            if (move_thread_flag_427 > 1):
              join move_thread_han_427
              $ 428 "Until (distance)"
              break
            end
            sync()
          end
          $ 429 "MoveJ"
          $ 430 "internos" "breakAfter"
          movej(internos, a=0.6981317007977318, v=0.5235987755982988)
          $ 431 "Wait: 0.3"
          sleep(0.3)
          $ 432 "Set CO[1]=Apagar"
          set_configurable_digital_out(1, False)
          $ 433 "Wait: 0.3"
          sleep(0.3)
          $ 434 "If barrenoActual≟13"
          if (barrenoActual == 13):
            $ 435 "Direction: Base Z+"
            global move_thread_flag_435=0
            thread move_thread_435():
              enter_critical
              move_thread_flag_435 = 1
              local towardsPos=calculate_point_to_move_towards(p[0.0,0.0,0.0,0.0,0.0,0.0], [0.0,0.0,1.0], 0.03)
              movel(towardsPos, a=1.2, v=0.25)
              move_thread_flag_435 = 2
              exit_critical
            end
            move_thread_flag_435 = 0
            move_thread_han_435 = run move_thread_435()
            while (True):
              sleep(1.0E-10)
              if (move_thread_flag_435 > 1):
                join move_thread_han_435
                $ 436 "Until (distance)"
                break
              end
              sync()
            end
            $ 437 "MoveJ"
            $ 438 "Zona_der1" "breakAfter"
            movej(get_inverse_kin(Zona_der1_p, qnear=Zona_der1_q), a=1.3962634015954636, v=1.0471975511965976)
            $ 439 "Posicion_Cero" "breakAfter"
            movej(get_inverse_kin(Posicion_Cero_p, qnear=Posicion_Cero_q), a=1.3962634015954636, v=1.0471975511965976)
            $ 440 "Call Quitar_Broca_Chida"
            Quitar_Broca_Chida()
            $ 441 "Call Poner_Broca"
            Poner_Broca()
            $ 442 "MoveJ"
            $ 443 "Posicion_Cero" "breakAfter"
            movej(get_inverse_kin(Posicion_Cero_p, qnear=Posicion_Cero_q), a=1.3962634015954636, v=1.0471975511965976)
            $ 444 "Zona_der1" "breakAfter"
            movej(get_inverse_kin(Zona_der1_p, qnear=Zona_der1_q), a=1.3962634015954636, v=1.0471975511965976)
          else:
            $ 445 "ElseIf barrenoActual≟27"
            if (barrenoActual == 27):
              $ 446 "Direction: Base Z+"
              global move_thread_flag_446=0
              thread move_thread_446():
                enter_critical
                move_thread_flag_446 = 1
                local towardsPos=calculate_point_to_move_towards(p[0.0,0.0,0.0,0.0,0.0,0.0], [0.0,0.0,1.0], 0.03)
                movel(towardsPos, a=1.2, v=0.25)
                move_thread_flag_446 = 2
                exit_critical
              end
              move_thread_flag_446 = 0
              move_thread_han_446 = run move_thread_446()
              while (True):
                sleep(1.0E-10)
                if (move_thread_flag_446 > 1):
                  join move_thread_han_446
                  $ 447 "Until (distance)"
                  break
                end
                sync()
              end
              $ 448 "MoveJ"
              $ 449 "Zona_der1" "breakAfter"
              movej(get_inverse_kin(Zona_der1_p, qnear=Zona_der1_q), a=1.3962634015954636, v=1.0471975511965976)
              $ 450 "Posicion_Cero" "breakAfter"
              movej(get_inverse_kin(Posicion_Cero_p, qnear=Posicion_Cero_q), a=1.3962634015954636, v=1.0471975511965976)
              $ 451 "Call Quitar_Broca_Chida"
              Quitar_Broca_Chida()
              $ 452 "Set carrusel_home=Encender"
              modbus_set_output_signal("carrusel_home", True)
              $ 453 "Wait: 1.0"
              sleep(1.0)
              $ 454 "Set carrusel_home=Apagar"
              modbus_set_output_signal("carrusel_home", False)
              $ 455 "Set mensaje_mw10=70"
              modbus_set_output_register("mensaje_mw10", 70)
              $ 456 "Wait Continuar_M30=HI"
              while (modbus_get_signal_status("Continuar_M30") == False):
                sync()
              end
              $ 457 "Wait: 1.0"
              sleep(1.0)
              $ 458 "Set mensaje_mw10=120"
              modbus_set_output_register("mensaje_mw10", 120)
              $ 459 "Wait Continuar_M30=HI"
              while (modbus_get_signal_status("Continuar_M30") == False):
                sync()
              end
              $ 460 "Wait: 1.0"
              sleep(1.0)
              $ 461 "Set carrusel_home=Encender"
              modbus_set_output_signal("carrusel_home", True)
              $ 462 "Wait: 1.0"
              sleep(1.0)
              $ 463 "Set carrusel_home=Apagar"
              modbus_set_output_signal("carrusel_home", False)
              $ 464 "Set mensaje_mw10=75"
              modbus_set_output_register("mensaje_mw10", 75)
              $ 465 "Wait Continuar_M30=HI"
              while (modbus_get_signal_status("Continuar_M30") == False):
                sync()
              end
              $ 466 "Wait: 1.0"
              sleep(1.0)
              $ 467 "Call Poner_Broca"
              Poner_Broca()
              $ 468 "broca≔1935"
              global broca=1935
              $ 469 "MoveJ"
              $ 470 "Posicion_Cero" "breakAfter"
              movej(get_inverse_kin(Posicion_Cero_p, qnear=Posicion_Cero_q), a=1.3962634015954636, v=1.0471975511965976)
              $ 471 "Zona_der1" "breakAfter"
              movej(get_inverse_kin(Zona_der1_p, qnear=Zona_der1_q), a=1.3962634015954636, v=1.0471975511965976)
              $ 472 "Set mensaje_mw10=80"
              modbus_set_output_register("mensaje_mw10", 80)
              $ 473 "Wait Continuar_M30=HI"
              while (modbus_get_signal_status("Continuar_M30") == False):
                sync()
              end
              $ 474 "Wait: 1.0"
              sleep(1.0)
              $ 475 "Set mensaje_mw10=150"
              modbus_set_output_register("mensaje_mw10", 150)
              $ 476 "Wait Continuar_M30=HI"
              while (modbus_get_signal_status("Continuar_M30") == False):
                sync()
              end
              $ 477 "Wait: 1.0"
              sleep(1.0)
            end
          end
          $ 478 "barrenoActual≔barrenoActual+1"
          global barrenoActual=barrenoActual+1
        end
        $ 479 "Linea 1 a 1935"
        $ 480 "broca≔1935"
        global broca=1935
        $ 481 "Buje_inicial"
        $ 482 "Buje_Inicial≔L1B2"
        global Buje_Inicial=L1B2
        $ 483 "Buje_final"
        $ 484 "Buje_Final≔L1B1"
        global Buje_Final=L1B1
        $ 485 "barrenosTotales≔27"
        global barrenosTotales=27
        $ 486 "barrenoActual≔1"
        global barrenoActual=1
        $ 487 "Loop barrenoActual≤barrenosTotales"
        while (barrenoActual <= barrenosTotales):
          $ 488 "MoveL"
          $ 489 "bajada_broca≔p[0,0,0.009,0,0,0]"
          global bajada_broca=p[0,0,0.009,0,0,0]
          $ 490 "internos≔interpolate_pose(Buje_Inicial, Buje_Final, ((barrenoActual)-1)/((barrenosTotales)-1))"
          global internos= interpolate_pose (Buje_Inicial, Buje_Final, ((barrenoActual)-1)/((barrenosTotales)-1))
          $ 491 "Alturas"
          $ 492 "If barrenoActual≟1 or barrenoActual≟3 or barrenoActual≟5 or barrenoActual≟7 or barrenoActual≟9 or barrenoActual≟11 or barrenoActual≟13 or barrenoActual≟15 or barrenoActual≟17 or barrenoActual≟19 or barrenoActual≟21 or barrenoActual≟23 or barrenoActual≟25 or barrenoActual≟27"
          if (barrenoActual == 1  or  barrenoActual == 3  or  barrenoActual == 5  or  barrenoActual == 7  or  barrenoActual == 9  or  barrenoActual == 11  or  barrenoActual == 13  or  barrenoActual == 15  or  barrenoActual == 17  or  barrenoActual == 19  or  barrenoActual == 21  or  barrenoActual == 23  or  barrenoActual == 25  or  barrenoActual == 27):
            $ 493 "Set mensaje_mw10=200"
            modbus_set_output_register("mensaje_mw10", 200)
            $ 494 "Wait Continuar_M30=HI"
            while (modbus_get_signal_status("Continuar_M30") == False):
              sync()
            end
            $ 495 "Wait: 1.0"
            sleep(1.0)
            $ 496 "Set mensaje_mw10=150"
            modbus_set_output_register("mensaje_mw10", 150)
            $ 497 "Wait: 1.0"
            sleep(1.0)
          end
          $ 498 "MoveJ"
          $ 499 "internos" "breakAfter"
          movej(internos, a=0.6981317007977318, v=0.5235987755982988)
          $ 500 "Wait: 2.0"
          sleep(2.0)
          $ 501 "If P1h[2]<P2h[2]"
          if (P1h[2]<P2h[2]):
            $ 502 "acomodo≔(altura/(barrenosTotales-1))*(barrenoActual-1)"
            global acomodo=(altura/(barrenosTotales-1))*(barrenoActual-1)
            $ 503 "tcp≔get_actual_tcp_pose()"
            global tcp= get_actual_tcp_pose ()
            $ 504 "offset_altura≔p[tcp[0],tcp[1],((alta-0.0095)-(acomodo/1000)),tcp[3],tcp[4],tcp[5]]"
            global offset_altura=p[tcp[0],tcp[1],((alta-0.0095)-(acomodo/1000)),tcp[3],tcp[4],tcp[5]]
            $ 505 "MoveL"
            $ 506 "offset_altura" "breakAfter"
            movel(offset_altura, a=0.04, v=0.03)
          else:
            $ 507 "Else" "noBreak"
            $ 508 "acomodo≔(altura/(barrenosTotales-1))*(26-(barrenoActual-1))"
            global acomodo=(altura/(barrenosTotales-1))*(26-(barrenoActual-1))
            $ 509 "tcp≔get_actual_tcp_pose()"
            global tcp= get_actual_tcp_pose ()
            $ 510 "offset_altura≔p[tcp[0],tcp[1],((alta-0.0095)-(acomodo/1000)),tcp[3],tcp[4],tcp[5]]"
            global offset_altura=p[tcp[0],tcp[1],((alta-0.0095)-(acomodo/1000)),tcp[3],tcp[4],tcp[5]]
            $ 511 "MoveL"
            $ 512 "offset_altura" "breakAfter"
            movel(offset_altura, a=0.04, v=0.03)
          end
          $ 513 "Freemove"
          $ 514 "Wait: 2.0"
          sleep(2.0)
          $ 515 "freedrive_mode()"
          freedrive_mode()
          $ 516 "Wait: 2.5"
          sleep(2.5)
          $ 517 "end_freedrive_mode()"
          end_freedrive_mode()
          $ 518 "Wait: 0.3"
          sleep(0.3)
          $ 519 "Set CO[1]=Encender"
          set_configurable_digital_out(1, True)
          $ 520 "Wait: 1.0"
          sleep(1.0)
          $ 521 "Wait: 0.3"
          sleep(0.3)
          $ 522 "Wait: 0.3"
          sleep(0.3)
          $ 523 "Wait: 0.3"
          sleep(0.3)
          $ 524 "Loop 2 times"
          Loop_63 = 0
          while (Loop_63 < 2):
            $ 525 "Poses_taladrado≔pose_sub(get_actual_tcp_pose(), bajada_broca)"
            global Poses_taladrado= pose_sub ( get_actual_tcp_pose (), bajada_broca)
            $ 526 "Poses_taladrado" "breakAfter"
            movel(Poses_taladrado, a=0.005, v=0.001)
            $ 527 "If bajada_broca≟p[0,0,0.018,0,0,0]"
            if (bajada_broca == p[0,0,0.018,0,0,0]):
              $ 528 "num_barreno≔str_cat('Barreno: ',barrenoActual)"
              global num_barreno=str_cat("Barreno: ",barrenoActual)
              $ 529 "tcp_actual≔get_actual_tcp_pose()"
              global tcp_actual= get_actual_tcp_pose ()
              $ 530 "X_actual≔str_cat('     X: ',tcp_actual[0])"
              global X_actual=str_cat("     X: ",tcp_actual[0])
              $ 531 "Y_actual≔str_cat('     Y: ',tcp_actual[1])"
              global Y_actual=str_cat("     Y: ",tcp_actual[1])
              $ 532 "pos_barreno≔str_cat(X_actual,Y_actual)"
              global pos_barreno=str_cat(X_actual,Y_actual)
              $ 533 "textmsg(num_barreno,pos_barreno)"
              textmsg(num_barreno,pos_barreno)
            end
            $ 534 "Poses_taladrado≔pose_add(get_actual_tcp_pose(), bajada_broca)"
            global Poses_taladrado= pose_add ( get_actual_tcp_pose (), bajada_broca)
            $ 535 "Poses_taladrado" "breakAfter"
            movel(Poses_taladrado, a=0.01, v=0.01)
            $ 536 "bajada_broca≔pose_add(bajada_broca, p[0,0,0.009,0,0,0])"
            global bajada_broca= pose_add (bajada_broca, p[0,0,0.009,0,0,0])
            Loop_63 = Loop_63 + 1
          end
          $ 537 "Direction: Base Z+"
          global move_thread_flag_537=0
          thread move_thread_537():
            enter_critical
            move_thread_flag_537 = 1
            local towardsPos=calculate_point_to_move_towards(p[0.0,0.0,0.0,0.0,0.0,0.0], [0.0,0.0,1.0], 0.05)
            movel(towardsPos, a=0.01, v=0.01)
            move_thread_flag_537 = 2
            exit_critical
          end
          move_thread_flag_537 = 0
          move_thread_han_537 = run move_thread_537()
          while (True):
            sleep(1.0E-10)
            if (move_thread_flag_537 > 1):
              join move_thread_han_537
              $ 538 "Until (distance)"
              break
            end
            sync()
          end
          $ 539 "MoveJ"
          $ 540 "internos" "breakAfter"
          movej(internos, a=0.6981317007977318, v=0.5235987755982988)
          $ 541 "Wait: 0.3"
          sleep(0.3)
          $ 542 "Set CO[1]=Apagar"
          set_configurable_digital_out(1, False)
          $ 543 "Wait: 0.3"
          sleep(0.3)
          $ 544 "If barrenoActual≟13 or barrenoActual≟27"
          if (barrenoActual == 13  or  barrenoActual == 27):
            $ 545 "Direction: Base Z+"
            global move_thread_flag_545=0
            thread move_thread_545():
              enter_critical
              move_thread_flag_545 = 1
              local towardsPos=calculate_point_to_move_towards(p[0.0,0.0,0.0,0.0,0.0,0.0], [0.0,0.0,1.0], 0.03)
              movel(towardsPos, a=0.04, v=0.03)
              move_thread_flag_545 = 2
              exit_critical
            end
            move_thread_flag_545 = 0
            move_thread_han_545 = run move_thread_545()
            while (True):
              sleep(1.0E-10)
              if (move_thread_flag_545 > 1):
                join move_thread_han_545
                $ 546 "Until (distance)"
                break
              end
              sync()
            end
            $ 547 "MoveJ"
            $ 548 "Zona_der1" "breakAfter"
            movej(get_inverse_kin(Zona_der1_p, qnear=Zona_der1_q), a=0.6981317007977318, v=0.5235987755982988)
            $ 549 "Posicion_Cero" "breakAfter"
            movej(get_inverse_kin(Posicion_Cero_p, qnear=Posicion_Cero_q), a=0.6981317007977318, v=0.5235987755982988)
            $ 550 "Call Quitar_Broca_Chida"
            Quitar_Broca_Chida()
            $ 551 "If barrenoActual≟13"
            if (barrenoActual == 13):
              $ 552 "Call Poner_Broca"
              Poner_Broca()
            else:
              $ 553 "ElseIf barrenoActual≟27"
              if (barrenoActual == 27):
                $ 554 "Call Poner_Broca"
                Poner_Broca()
              end
            end
            $ 555 "MoveJ"
            $ 556 "Posicion_Cero" "breakAfter"
            movej(get_inverse_kin(Posicion_Cero_p, qnear=Posicion_Cero_q), a=0.6981317007977318, v=0.5235987755982988)
            $ 557 "Zona_der1" "breakAfter"
            movej(get_inverse_kin(Zona_der1_p, qnear=Zona_der1_q), a=0.6981317007977318, v=0.5235987755982988)
          end
          $ 558 "barrenoActual≔barrenoActual+1"
          global barrenoActual=barrenoActual+1
        end
        $ 559 "Linea 2 a 1935"
        $ 560 "broca≔1935"
        global broca=1935
        $ 561 "Buje_inicial"
        $ 562 "Buje_Inicial≔L2B2"
        global Buje_Inicial=L2B2
        $ 563 "Buje_final"
        $ 564 "Buje_Final≔L2B1"
        global Buje_Final=L2B1
        $ 565 "barrenosTotales≔27"
        global barrenosTotales=27
        $ 566 "barrenoActual≔1"
        global barrenoActual=1
        $ 567 "Loop barrenoActual≤barrenosTotales"
        while (barrenoActual <= barrenosTotales):
          $ 568 "MoveL"
          $ 569 "bajada_broca≔p[0,0,0.009,0,0,0]"
          global bajada_broca=p[0,0,0.009,0,0,0]
          $ 570 "internos≔interpolate_pose(Buje_Inicial, Buje_Final, ((barrenoActual)-1)/((barrenosTotales)-1))"
          global internos= interpolate_pose (Buje_Inicial, Buje_Final, ((barrenoActual)-1)/((barrenosTotales)-1))
          $ 571 "Alturas"
          $ 572 "If barrenoActual≟1 or barrenoActual≟3 or barrenoActual≟5 or barrenoActual≟7 or barrenoActual≟9 or barrenoActual≟11 or barrenoActual≟13 or barrenoActual≟15 or barrenoActual≟17 or barrenoActual≟19 or barrenoActual≟21 or barrenoActual≟23 or barrenoActual≟25 or barrenoActual≟27"
          if (barrenoActual == 1  or  barrenoActual == 3  or  barrenoActual == 5  or  barrenoActual == 7  or  barrenoActual == 9  or  barrenoActual == 11  or  barrenoActual == 13  or  barrenoActual == 15  or  barrenoActual == 17  or  barrenoActual == 19  or  barrenoActual == 21  or  barrenoActual == 23  or  barrenoActual == 25  or  barrenoActual == 27):
            $ 573 "Set mensaje_mw10=200"
            modbus_set_output_register("mensaje_mw10", 200)
            $ 574 "Wait Continuar_M30=HI"
            while (modbus_get_signal_status("Continuar_M30") == False):
              sync()
            end
            $ 575 "Wait: 1.0"
            sleep(1.0)
            $ 576 "Set mensaje_mw10=150"
            modbus_set_output_register("mensaje_mw10", 150)
            $ 577 "Wait: 1.0"
            sleep(1.0)
          end
          $ 578 "MoveJ"
          $ 579 "internos" "breakAfter"
          movej(internos, a=0.6981317007977318, v=0.5235987755982988)
          $ 580 "Wait: 2.0"
          sleep(2.0)
          $ 581 "If P1h[2]<P2h[2]"
          if (P1h[2]<P2h[2]):
            $ 582 "acomodo≔(altura/(barrenosTotales-1))*(barrenoActual-1)"
            global acomodo=(altura/(barrenosTotales-1))*(barrenoActual-1)
            $ 583 "tcp≔get_actual_tcp_pose()"
            global tcp= get_actual_tcp_pose ()
            $ 584 "offset_altura≔p[tcp[0],tcp[1],((alta-0.0095)-(acomodo/1000)),tcp[3],tcp[4],tcp[5]]"
            global offset_altura=p[tcp[0],tcp[1],((alta-0.0095)-(acomodo/1000)),tcp[3],tcp[4],tcp[5]]
            $ 585 "MoveL"
            $ 586 "offset_altura" "breakAfter"
            movel(offset_altura, a=0.04, v=0.03)
          else:
            $ 587 "Else" "noBreak"
            $ 588 "acomodo≔(altura/(barrenosTotales-1))*(26-(barrenoActual-1))"
            global acomodo=(altura/(barrenosTotales-1))*(26-(barrenoActual-1))
            $ 589 "tcp≔get_actual_tcp_pose()"
            global tcp= get_actual_tcp_pose ()
            $ 590 "offset_altura≔p[tcp[0],tcp[1],((alta-0.0095)-(acomodo/1000)),tcp[3],tcp[4],tcp[5]]"
            global offset_altura=p[tcp[0],tcp[1],((alta-0.0095)-(acomodo/1000)),tcp[3],tcp[4],tcp[5]]
            $ 591 "MoveL"
            $ 592 "offset_altura" "breakAfter"
            movel(offset_altura, a=0.04, v=0.03)
          end
          $ 593 "Freemove"
          $ 594 "Wait: 2.0"
          sleep(2.0)
          $ 595 "freedrive_mode()"
          freedrive_mode()
          $ 596 "Wait: 2.5"
          sleep(2.5)
          $ 597 "end_freedrive_mode()"
          end_freedrive_mode()
          $ 598 "Wait: 0.3"
          sleep(0.3)
          $ 599 "Set CO[1]=Encender"
          set_configurable_digital_out(1, True)
          $ 600 "Wait: 1.0"
          sleep(1.0)
          $ 601 "Wait: 0.3"
          sleep(0.3)
          $ 602 "Wait: 0.3"
          sleep(0.3)
          $ 603 "Wait: 0.3"
          sleep(0.3)
          $ 604 "Loop 2 times"
          Loop_65 = 0
          while (Loop_65 < 2):
            $ 605 "Poses_taladrado≔pose_sub(get_actual_tcp_pose(), bajada_broca)"
            global Poses_taladrado= pose_sub ( get_actual_tcp_pose (), bajada_broca)
            $ 606 "Poses_taladrado" "breakAfter"
            movel(Poses_taladrado, a=0.005, v=0.001)
            $ 607 "If bajada_broca≟p[0,0,0.018,0,0,0]"
            if (bajada_broca == p[0,0,0.018,0,0,0]):
              $ 608 "num_barreno≔str_cat('Barreno: ',barrenoActual)"
              global num_barreno=str_cat("Barreno: ",barrenoActual)
              $ 609 "tcp_actual≔get_actual_tcp_pose()"
              global tcp_actual= get_actual_tcp_pose ()
              $ 610 "X_actual≔str_cat('     X: ',tcp_actual[0])"
              global X_actual=str_cat("     X: ",tcp_actual[0])
              $ 611 "Y_actual≔str_cat('     Y: ',tcp_actual[1])"
              global Y_actual=str_cat("     Y: ",tcp_actual[1])
              $ 612 "pos_barreno≔str_cat(X_actual,Y_actual)"
              global pos_barreno=str_cat(X_actual,Y_actual)
              $ 613 "textmsg(num_barreno,pos_barreno)"
              textmsg(num_barreno,pos_barreno)
            end
            $ 614 "Poses_taladrado≔pose_add(get_actual_tcp_pose(), bajada_broca)"
            global Poses_taladrado= pose_add ( get_actual_tcp_pose (), bajada_broca)
            $ 615 "Poses_taladrado" "breakAfter"
            movel(Poses_taladrado, a=0.01, v=0.01)
            $ 616 "bajada_broca≔pose_add(bajada_broca, p[0,0,0.009,0,0,0])"
            global bajada_broca= pose_add (bajada_broca, p[0,0,0.009,0,0,0])
            Loop_65 = Loop_65 + 1
          end
          $ 617 "Direction: Base Z+"
          global move_thread_flag_617=0
          thread move_thread_617():
            enter_critical
            move_thread_flag_617 = 1
            local towardsPos=calculate_point_to_move_towards(p[0.0,0.0,0.0,0.0,0.0,0.0], [0.0,0.0,1.0], 0.05)
            movel(towardsPos, a=0.01, v=0.01)
            move_thread_flag_617 = 2
            exit_critical
          end
          move_thread_flag_617 = 0
          move_thread_han_617 = run move_thread_617()
          while (True):
            sleep(1.0E-10)
            if (move_thread_flag_617 > 1):
              join move_thread_han_617
              $ 618 "Until (distance)"
              break
            end
            sync()
          end
          $ 619 "MoveJ"
          $ 620 "internos" "breakAfter"
          movej(internos, a=0.6981317007977318, v=0.5235987755982988)
          $ 621 "Wait: 0.3"
          sleep(0.3)
          $ 622 "Set CO[1]=Apagar"
          set_configurable_digital_out(1, False)
          $ 623 "Wait: 0.3"
          sleep(0.3)
          $ 624 "If barrenoActual≟13"
          if (barrenoActual == 13):
            $ 625 "Direction: Base Z+"
            global move_thread_flag_625=0
            thread move_thread_625():
              enter_critical
              move_thread_flag_625 = 1
              local towardsPos=calculate_point_to_move_towards(p[0.0,0.0,0.0,0.0,0.0,0.0], [0.0,0.0,1.0], 0.03)
              movel(towardsPos, a=0.04, v=0.03)
              move_thread_flag_625 = 2
              exit_critical
            end
            move_thread_flag_625 = 0
            move_thread_han_625 = run move_thread_625()
            while (True):
              sleep(1.0E-10)
              if (move_thread_flag_625 > 1):
                join move_thread_han_625
                $ 626 "Until (distance)"
                break
              end
              sync()
            end
            $ 627 "MoveJ"
            $ 628 "Zona_der1" "breakAfter"
            movej(get_inverse_kin(Zona_der1_p, qnear=Zona_der1_q), a=1.3962634015954636, v=1.0471975511965976)
            $ 629 "Posicion_Cero" "breakAfter"
            movej(get_inverse_kin(Posicion_Cero_p, qnear=Posicion_Cero_q), a=1.3962634015954636, v=1.0471975511965976)
            $ 630 "Call Quitar_Broca_Chida"
            Quitar_Broca_Chida()
            $ 631 "Call Poner_Broca"
            Poner_Broca()
            $ 632 "MoveJ"
            $ 633 "Posicion_Cero" "breakAfter"
            movej(get_inverse_kin(Posicion_Cero_p, qnear=Posicion_Cero_q), a=1.3962634015954636, v=1.0471975511965976)
            $ 634 "Zona_der1" "breakAfter"
            movej(get_inverse_kin(Zona_der1_p, qnear=Zona_der1_q), a=1.3962634015954636, v=1.0471975511965976)
          else:
            $ 635 "ElseIf barrenoActual≟27"
            if (barrenoActual == 27):
              $ 636 "Direction: Base Z+"
              global move_thread_flag_636=0
              thread move_thread_636():
                enter_critical
                move_thread_flag_636 = 1
                local towardsPos=calculate_point_to_move_towards(p[0.0,0.0,0.0,0.0,0.0,0.0], [0.0,0.0,1.0], 0.03)
                movel(towardsPos, a=0.04, v=0.03)
                move_thread_flag_636 = 2
                exit_critical
              end
              move_thread_flag_636 = 0
              move_thread_han_636 = run move_thread_636()
              while (True):
                sleep(1.0E-10)
                if (move_thread_flag_636 > 1):
                  join move_thread_han_636
                  $ 637 "Until (distance)"
                  break
                end
                sync()
              end
              $ 638 "MoveJ"
              $ 639 "Zona_der1" "breakAfter"
              movej(get_inverse_kin(Zona_der1_p, qnear=Zona_der1_q), a=1.3962634015954636, v=1.0471975511965976)
              $ 640 "Posicion_Cero" "breakAfter"
              movej(get_inverse_kin(Posicion_Cero_p, qnear=Posicion_Cero_q), a=1.3962634015954636, v=1.0471975511965976)
              $ 641 "Call Quitar_Broca_Chida"
              Quitar_Broca_Chida()
              $ 642 "Set carrusel_home=Encender"
              modbus_set_output_signal("carrusel_home", True)
              $ 643 "Wait: 1.0"
              sleep(1.0)
              $ 644 "Set carrusel_home=Apagar"
              modbus_set_output_signal("carrusel_home", False)
              $ 645 "Set mensaje_mw10=85"
              modbus_set_output_register("mensaje_mw10", 85)
              $ 646 "Wait Continuar_M30=HI"
              while (modbus_get_signal_status("Continuar_M30") == False):
                sync()
              end
              $ 647 "Wait: 1.0"
              sleep(1.0)
              $ 648 "Set mensaje_mw10=120"
              modbus_set_output_register("mensaje_mw10", 120)
              $ 649 "Wait Continuar_M30=HI"
              while (modbus_get_signal_status("Continuar_M30") == False):
                sync()
              end
              $ 650 "Wait: 1.0"
              sleep(1.0)
              $ 651 "Set carrusel_home=Encender"
              modbus_set_output_signal("carrusel_home", True)
              $ 652 "Wait: 1.0"
              sleep(1.0)
              $ 653 "Set carrusel_home=Apagar"
              modbus_set_output_signal("carrusel_home", False)
              $ 654 "Set mensaje_mw10=90"
              modbus_set_output_register("mensaje_mw10", 90)
              $ 655 "Wait Continuar_M30=HI"
              while (modbus_get_signal_status("Continuar_M30") == False):
                sync()
              end
              $ 656 "Wait: 1.0"
              sleep(1.0)
              $ 657 "Call Poner_Broca"
              Poner_Broca()
              $ 658 "broca≔217"
              global broca=217
              $ 659 "MoveJ"
              $ 660 "Posicion_Cero" "breakAfter"
              movej(get_inverse_kin(Posicion_Cero_p, qnear=Posicion_Cero_q), a=1.3962634015954636, v=1.0471975511965976)
              $ 661 "Zona_der1" "breakAfter"
              movej(get_inverse_kin(Zona_der1_p, qnear=Zona_der1_q), a=1.3962634015954636, v=1.0471975511965976)
              $ 662 "Set mensaje_mw10=95"
              modbus_set_output_register("mensaje_mw10", 95)
              $ 663 "Wait Continuar_M30=HI"
              while (modbus_get_signal_status("Continuar_M30") == False):
                sync()
              end
              $ 664 "Wait: 1.0"
              sleep(1.0)
              $ 665 "Set mensaje_mw10=150"
              modbus_set_output_register("mensaje_mw10", 150)
              $ 666 "Wait Continuar_M30=HI"
              while (modbus_get_signal_status("Continuar_M30") == False):
                sync()
              end
              $ 667 "Wait: 1.0"
              sleep(1.0)
            end
          end
          $ 668 "barrenoActual≔barrenoActual+1"
          global barrenoActual=barrenoActual+1
        end
        $ 669 "Linea 1 a 217"
        $ 670 "broca≔217"
        global broca=217
        $ 671 "Buje_inicial"
        $ 672 "Buje_Inicial≔L1B2"
        global Buje_Inicial=L1B2
        $ 673 "Buje_final"
        $ 674 "Buje_Final≔L1B1"
        global Buje_Final=L1B1
        $ 675 "barrenosTotales≔27"
        global barrenosTotales=27
        $ 676 "barrenoActual≔1"
        global barrenoActual=1
        $ 677 "Loop barrenoActual≤barrenosTotales"
        while (barrenoActual <= barrenosTotales):
          $ 678 "MoveL"
          $ 679 "bajada_broca≔p[0,0,0.018,0,0,0]"
          global bajada_broca=p[0,0,0.018,0,0,0]
          $ 680 "internos≔interpolate_pose(Buje_Inicial, Buje_Final, ((barrenoActual)-1)/((barrenosTotales)-1))"
          global internos= interpolate_pose (Buje_Inicial, Buje_Final, ((barrenoActual)-1)/((barrenosTotales)-1))
          $ 681 "Wait: 2.0"
          sleep(2.0)
          $ 682 "Alturas"
          $ 683 "If barrenoActual≟1 or barrenoActual≟3 or barrenoActual≟5 or barrenoActual≟7 or barrenoActual≟9 or barrenoActual≟11 or barrenoActual≟13 or barrenoActual≟15 or barrenoActual≟17 or barrenoActual≟19 or barrenoActual≟21 or barrenoActual≟23 or barrenoActual≟25 or barrenoActual≟27"
          if (barrenoActual == 1  or  barrenoActual == 3  or  barrenoActual == 5  or  barrenoActual == 7  or  barrenoActual == 9  or  barrenoActual == 11  or  barrenoActual == 13  or  barrenoActual == 15  or  barrenoActual == 17  or  barrenoActual == 19  or  barrenoActual == 21  or  barrenoActual == 23  or  barrenoActual == 25  or  barrenoActual == 27):
            $ 684 "Set mensaje_mw10=200"
            modbus_set_output_register("mensaje_mw10", 200)
            $ 685 "Wait Continuar_M30=HI"
            while (modbus_get_signal_status("Continuar_M30") == False):
              sync()
            end
            $ 686 "Wait: 1.0"
            sleep(1.0)
            $ 687 "Set mensaje_mw10=150"
            modbus_set_output_register("mensaje_mw10", 150)
            $ 688 "Wait: 1.0"
            sleep(1.0)
          end
          $ 689 "MoveJ"
          $ 690 "internos" "breakAfter"
          movej(internos, a=0.6981317007977318, v=0.5235987755982988)
          $ 691 "Wait: 2.0"
          sleep(2.0)
          $ 692 "If P1h[2]<P2h[2]"
          if (P1h[2]<P2h[2]):
            $ 693 "acomodo≔(altura/(barrenosTotales-1))*(barrenoActual-1)"
            global acomodo=(altura/(barrenosTotales-1))*(barrenoActual-1)
            $ 694 "tcp≔get_actual_tcp_pose()"
            global tcp= get_actual_tcp_pose ()
            $ 695 "offset_altura≔p[tcp[0],tcp[1],((alta-0.0095)-(acomodo/1000)),tcp[3],tcp[4],tcp[5]]"
            global offset_altura=p[tcp[0],tcp[1],((alta-0.0095)-(acomodo/1000)),tcp[3],tcp[4],tcp[5]]
            $ 696 "MoveL"
            $ 697 "offset_altura" "breakAfter"
            movel(offset_altura, a=0.04, v=0.03)
          else:
            $ 698 "Else" "noBreak"
            $ 699 "acomodo≔(altura/(barrenosTotales-1))*(26-(barrenoActual-1))"
            global acomodo=(altura/(barrenosTotales-1))*(26-(barrenoActual-1))
            $ 700 "tcp≔get_actual_tcp_pose()"
            global tcp= get_actual_tcp_pose ()
            $ 701 "offset_altura≔p[tcp[0],tcp[1],((alta-0.0095)-(acomodo/1000)),tcp[3],tcp[4],tcp[5]]"
            global offset_altura=p[tcp[0],tcp[1],((alta-0.0095)-(acomodo/1000)),tcp[3],tcp[4],tcp[5]]
            $ 702 "MoveL"
            $ 703 "offset_altura" "breakAfter"
            movel(offset_altura, a=0.04, v=0.03)
          end
          $ 704 "Freemove"
          $ 705 "Wait: 2.0"
          sleep(2.0)
          $ 706 "freedrive_mode()"
          freedrive_mode()
          $ 707 "Wait: 2.5"
          sleep(2.5)
          $ 708 "end_freedrive_mode()"
          end_freedrive_mode()
          $ 709 "Wait: 0.3"
          sleep(0.3)
          $ 710 "Set CO[1]=Encender"
          set_configurable_digital_out(1, True)
          $ 711 "Wait: 1.0"
          sleep(1.0)
          $ 712 "Wait: 0.3"
          sleep(0.3)
          $ 713 "Wait: 0.3"
          sleep(0.3)
          $ 714 "Wait: 0.3"
          sleep(0.3)
          $ 715 "Loop 1 times"
          Loop_67 = 0
          while (Loop_67 < 1):
            $ 716 "Poses_taladrado≔pose_sub(get_actual_tcp_pose(), bajada_broca)"
            global Poses_taladrado= pose_sub ( get_actual_tcp_pose (), bajada_broca)
            $ 717 "Poses_taladrado" "breakAfter"
            movel(Poses_taladrado, a=0.005, v=0.001)
            $ 718 "If bajada_broca≟p[0,0,0.018,0,0,0]"
            if (bajada_broca == p[0,0,0.018,0,0,0]):
              $ 719 "num_barreno≔str_cat('Barreno: ',barrenoActual)"
              global num_barreno=str_cat("Barreno: ",barrenoActual)
              $ 720 "tcp_actual≔get_actual_tcp_pose()"
              global tcp_actual= get_actual_tcp_pose ()
              $ 721 "X_actual≔str_cat('     X: ',tcp_actual[0])"
              global X_actual=str_cat("     X: ",tcp_actual[0])
              $ 722 "Y_actual≔str_cat('     Y: ',tcp_actual[1])"
              global Y_actual=str_cat("     Y: ",tcp_actual[1])
              $ 723 "pos_barreno≔str_cat(X_actual,Y_actual)"
              global pos_barreno=str_cat(X_actual,Y_actual)
              $ 724 "textmsg(num_barreno,pos_barreno)"
              textmsg(num_barreno,pos_barreno)
            end
            $ 725 "Poses_taladrado≔pose_add(get_actual_tcp_pose(), bajada_broca)"
            global Poses_taladrado= pose_add ( get_actual_tcp_pose (), bajada_broca)
            $ 726 "Poses_taladrado" "breakAfter"
            movel(Poses_taladrado, a=0.01, v=0.01)
            $ 727 "bajada_broca≔pose_add(bajada_broca, p[0,0,0.018,0,0,0])"
            global bajada_broca= pose_add (bajada_broca, p[0,0,0.018,0,0,0])
            Loop_67 = Loop_67 + 1
          end
          $ 728 "Direction: Base Z+"
          global move_thread_flag_728=0
          thread move_thread_728():
            enter_critical
            move_thread_flag_728 = 1
            local towardsPos=calculate_point_to_move_towards(p[0.0,0.0,0.0,0.0,0.0,0.0], [0.0,0.0,1.0], 0.05)
            movel(towardsPos, a=0.01, v=0.01)
            move_thread_flag_728 = 2
            exit_critical
          end
          move_thread_flag_728 = 0
          move_thread_han_728 = run move_thread_728()
          while (True):
            sleep(1.0E-10)
            if (move_thread_flag_728 > 1):
              join move_thread_han_728
              $ 729 "Until (distance)"
              break
            end
            sync()
          end
          $ 730 "MoveJ"
          $ 731 "internos" "breakAfter"
          movej(internos, a=0.6981317007977318, v=0.5235987755982988)
          $ 732 "Wait: 0.3"
          sleep(0.3)
          $ 733 "Set CO[1]=Apagar"
          set_configurable_digital_out(1, False)
          $ 734 "Wait: 0.3"
          sleep(0.3)
          $ 735 "If barrenoActual≟13 or barrenoActual≟27"
          if (barrenoActual == 13  or  barrenoActual == 27):
            $ 736 "Direction: Base Z+"
            global move_thread_flag_736=0
            thread move_thread_736():
              enter_critical
              move_thread_flag_736 = 1
              local towardsPos=calculate_point_to_move_towards(p[0.0,0.0,0.0,0.0,0.0,0.0], [0.0,0.0,1.0], 0.03)
              movel(towardsPos, a=0.03, v=0.04)
              move_thread_flag_736 = 2
              exit_critical
            end
            move_thread_flag_736 = 0
            move_thread_han_736 = run move_thread_736()
            while (True):
              sleep(1.0E-10)
              if (move_thread_flag_736 > 1):
                join move_thread_han_736
                $ 737 "Until (distance)"
                break
              end
              sync()
            end
            $ 738 "MoveJ"
            $ 739 "Zona_der1" "breakAfter"
            movej(get_inverse_kin(Zona_der1_p, qnear=Zona_der1_q), a=0.6981317007977318, v=0.5235987755982988)
            $ 740 "Posicion_Cero" "breakAfter"
            movej(get_inverse_kin(Posicion_Cero_p, qnear=Posicion_Cero_q), a=0.6981317007977318, v=0.5235987755982988)
            $ 741 "Call Quitar_Broca_Chida"
            Quitar_Broca_Chida()
            $ 742 "If barrenoActual≟13"
            if (barrenoActual == 13):
              $ 743 "Call Poner_Broca"
              Poner_Broca()
            else:
              $ 744 "ElseIf barrenoActual≟27"
              if (barrenoActual == 27):
                $ 745 "Call Poner_Broca"
                Poner_Broca()
              end
            end
            $ 746 "MoveJ"
            $ 747 "Posicion_Cero" "breakAfter"
            movej(get_inverse_kin(Posicion_Cero_p, qnear=Posicion_Cero_q), a=0.6981317007977318, v=0.5235987755982988)
            $ 748 "Zona_der1" "breakAfter"
            movej(get_inverse_kin(Zona_der1_p, qnear=Zona_der1_q), a=0.6981317007977318, v=0.5235987755982988)
          end
          $ 749 "barrenoActual≔barrenoActual+1"
          global barrenoActual=barrenoActual+1
        end
        $ 750 "Linea 2 a 217"
        $ 751 "broca≔217"
        global broca=217
        $ 752 "Buje_inicial"
        $ 753 "Buje_Inicial≔L2B2"
        global Buje_Inicial=L2B2
        $ 754 "Buje_final"
        $ 755 "Buje_Final≔L2B1"
        global Buje_Final=L2B1
        $ 756 "barrenosTotales≔27"
        global barrenosTotales=27
        $ 757 "barrenoActual≔1"
        global barrenoActual=1
        $ 758 "Loop barrenoActual≤barrenosTotales"
        while (barrenoActual <= barrenosTotales):
          $ 759 "MoveL"
          $ 760 "bajada_broca≔p[0,0,0.018,0,0,0]"
          global bajada_broca=p[0,0,0.018,0,0,0]
          $ 761 "internos≔interpolate_pose(Buje_Inicial, Buje_Final, ((barrenoActual)-1)/((barrenosTotales)-1))"
          global internos= interpolate_pose (Buje_Inicial, Buje_Final, ((barrenoActual)-1)/((barrenosTotales)-1))
          $ 762 "Alturas"
          $ 763 "If barrenoActual≟1 or barrenoActual≟3 or barrenoActual≟5 or barrenoActual≟7 or barrenoActual≟9 or barrenoActual≟11 or barrenoActual≟13 or barrenoActual≟15 or barrenoActual≟17 or barrenoActual≟19 or barrenoActual≟21 or barrenoActual≟23 or barrenoActual≟25 or barrenoActual≟27"
          if (barrenoActual == 1  or  barrenoActual == 3  or  barrenoActual == 5  or  barrenoActual == 7  or  barrenoActual == 9  or  barrenoActual == 11  or  barrenoActual == 13  or  barrenoActual == 15  or  barrenoActual == 17  or  barrenoActual == 19  or  barrenoActual == 21  or  barrenoActual == 23  or  barrenoActual == 25  or  barrenoActual == 27):
            $ 764 "Set mensaje_mw10=200"
            modbus_set_output_register("mensaje_mw10", 200)
            $ 765 "Wait Continuar_M30=HI"
            while (modbus_get_signal_status("Continuar_M30") == False):
              sync()
            end
            $ 766 "Wait: 1.0"
            sleep(1.0)
            $ 767 "Set mensaje_mw10=150"
            modbus_set_output_register("mensaje_mw10", 150)
            $ 768 "Wait: 1.0"
            sleep(1.0)
          end
          $ 769 "MoveJ"
          $ 770 "internos" "breakAfter"
          movej(internos, a=0.6981317007977318, v=0.5235987755982988)
          $ 771 "Wait: 2.0"
          sleep(2.0)
          $ 772 "If P1h[2]<P2h[2]"
          if (P1h[2]<P2h[2]):
            $ 773 "acomodo≔(altura/(barrenosTotales-1))*(barrenoActual-1)"
            global acomodo=(altura/(barrenosTotales-1))*(barrenoActual-1)
            $ 774 "tcp≔get_actual_tcp_pose()"
            global tcp= get_actual_tcp_pose ()
            $ 775 "offset_altura≔p[tcp[0],tcp[1],((alta-0.0095)-(acomodo/1000)),tcp[3],tcp[4],tcp[5]]"
            global offset_altura=p[tcp[0],tcp[1],((alta-0.0095)-(acomodo/1000)),tcp[3],tcp[4],tcp[5]]
            $ 776 "MoveL"
            $ 777 "offset_altura" "breakAfter"
            movel(offset_altura, a=0.04, v=0.03)
          else:
            $ 778 "Else" "noBreak"
            $ 779 "acomodo≔(altura/(barrenosTotales-1))*(26-(barrenoActual-1))"
            global acomodo=(altura/(barrenosTotales-1))*(26-(barrenoActual-1))
            $ 780 "tcp≔get_actual_tcp_pose()"
            global tcp= get_actual_tcp_pose ()
            $ 781 "offset_altura≔p[tcp[0],tcp[1],((alta-0.0095)-(acomodo/1000)),tcp[3],tcp[4],tcp[5]]"
            global offset_altura=p[tcp[0],tcp[1],((alta-0.0095)-(acomodo/1000)),tcp[3],tcp[4],tcp[5]]
            $ 782 "MoveL"
            $ 783 "offset_altura" "breakAfter"
            movel(offset_altura, a=0.04, v=0.03)
          end
          $ 784 "Freemove"
          $ 785 "Wait: 2.0"
          sleep(2.0)
          $ 786 "freedrive_mode()"
          freedrive_mode()
          $ 787 "Wait: 2.5"
          sleep(2.5)
          $ 788 "end_freedrive_mode()"
          end_freedrive_mode()
          $ 789 "Wait: 0.3"
          sleep(0.3)
          $ 790 "Set CO[1]=Encender"
          set_configurable_digital_out(1, True)
          $ 791 "Wait: 1.0"
          sleep(1.0)
          $ 792 "Wait: 0.3"
          sleep(0.3)
          $ 793 "Wait: 0.3"
          sleep(0.3)
          $ 794 "Wait: 0.3"
          sleep(0.3)
          $ 795 "Loop 1 times"
          Loop_69 = 0
          while (Loop_69 < 1):
            $ 796 "Poses_taladrado≔pose_sub(get_actual_tcp_pose(), bajada_broca)"
            global Poses_taladrado= pose_sub ( get_actual_tcp_pose (), bajada_broca)
            $ 797 "Poses_taladrado" "breakAfter"
            movel(Poses_taladrado, a=0.005, v=0.001)
            $ 798 "If bajada_broca≟p[0,0,0.018,0,0,0]"
            if (bajada_broca == p[0,0,0.018,0,0,0]):
              $ 799 "num_barreno≔str_cat('Barreno: ',barrenoActual)"
              global num_barreno=str_cat("Barreno: ",barrenoActual)
              $ 800 "tcp_actual≔get_actual_tcp_pose()"
              global tcp_actual= get_actual_tcp_pose ()
              $ 801 "X_actual≔str_cat('     X: ',tcp_actual[0])"
              global X_actual=str_cat("     X: ",tcp_actual[0])
              $ 802 "Y_actual≔str_cat('     Y: ',tcp_actual[1])"
              global Y_actual=str_cat("     Y: ",tcp_actual[1])
              $ 803 "pos_barreno≔str_cat(X_actual,Y_actual)"
              global pos_barreno=str_cat(X_actual,Y_actual)
              $ 804 "textmsg(num_barreno,pos_barreno)"
              textmsg(num_barreno,pos_barreno)
            end
            $ 805 "Poses_taladrado≔pose_add(get_actual_tcp_pose(), bajada_broca)"
            global Poses_taladrado= pose_add ( get_actual_tcp_pose (), bajada_broca)
            $ 806 "Poses_taladrado" "breakAfter"
            movel(Poses_taladrado, a=0.01, v=0.01)
            $ 807 "bajada_broca≔pose_add(bajada_broca, p[0,0,0.018,0,0,0])"
            global bajada_broca= pose_add (bajada_broca, p[0,0,0.018,0,0,0])
            Loop_69 = Loop_69 + 1
          end
          $ 808 "Direction: Base Z+"
          global move_thread_flag_808=0
          thread move_thread_808():
            enter_critical
            move_thread_flag_808 = 1
            local towardsPos=calculate_point_to_move_towards(p[0.0,0.0,0.0,0.0,0.0,0.0], [0.0,0.0,1.0], 0.05)
            movel(towardsPos, a=0.01, v=0.01)
            move_thread_flag_808 = 2
            exit_critical
          end
          move_thread_flag_808 = 0
          move_thread_han_808 = run move_thread_808()
          while (True):
            sleep(1.0E-10)
            if (move_thread_flag_808 > 1):
              join move_thread_han_808
              $ 809 "Until (distance)"
              break
            end
            sync()
          end
          $ 810 "MoveJ"
          $ 811 "internos" "breakAfter"
          movej(internos, a=0.6981317007977318, v=0.5235987755982988)
          $ 812 "Wait: 0.3"
          sleep(0.3)
          $ 813 "Set CO[1]=Apagar"
          set_configurable_digital_out(1, False)
          $ 814 "Wait: 0.3"
          sleep(0.3)
          $ 815 "If barrenoActual≟13"
          if (barrenoActual == 13):
            $ 816 "Direction: Base Z+"
            global move_thread_flag_816=0
            thread move_thread_816():
              enter_critical
              move_thread_flag_816 = 1
              local towardsPos=calculate_point_to_move_towards(p[0.0,0.0,0.0,0.0,0.0,0.0], [0.0,0.0,1.0], 0.03)
              movel(towardsPos, a=0.04, v=0.03)
              move_thread_flag_816 = 2
              exit_critical
            end
            move_thread_flag_816 = 0
            move_thread_han_816 = run move_thread_816()
            while (True):
              sleep(1.0E-10)
              if (move_thread_flag_816 > 1):
                join move_thread_han_816
                $ 817 "Until (distance)"
                break
              end
              sync()
            end
            $ 818 "MoveJ"
            $ 819 "Zona_der1" "breakAfter"
            movej(get_inverse_kin(Zona_der1_p, qnear=Zona_der1_q), a=1.3962634015954636, v=1.0471975511965976)
            $ 820 "Posicion_Cero" "breakAfter"
            movej(get_inverse_kin(Posicion_Cero_p, qnear=Posicion_Cero_q), a=1.3962634015954636, v=1.0471975511965976)
            $ 821 "Call Quitar_Broca_Chida"
            Quitar_Broca_Chida()
            $ 822 "Call Poner_Broca"
            Poner_Broca()
            $ 823 "MoveJ"
            $ 824 "Posicion_Cero" "breakAfter"
            movej(get_inverse_kin(Posicion_Cero_p, qnear=Posicion_Cero_q), a=1.3962634015954636, v=1.0471975511965976)
            $ 825 "Zona_der1" "breakAfter"
            movej(get_inverse_kin(Zona_der1_p, qnear=Zona_der1_q), a=1.3962634015954636, v=1.0471975511965976)
          else:
            $ 826 "ElseIf barrenoActual≟27"
            if (barrenoActual == 27):
              $ 827 "Direction: Base Z+"
              global move_thread_flag_827=0
              thread move_thread_827():
                enter_critical
                move_thread_flag_827 = 1
                local towardsPos=calculate_point_to_move_towards(p[0.0,0.0,0.0,0.0,0.0,0.0], [0.0,0.0,1.0], 0.03)
                movel(towardsPos, a=0.04, v=0.03)
                move_thread_flag_827 = 2
                exit_critical
              end
              move_thread_flag_827 = 0
              move_thread_han_827 = run move_thread_827()
              while (True):
                sleep(1.0E-10)
                if (move_thread_flag_827 > 1):
                  join move_thread_han_827
                  $ 828 "Until (distance)"
                  break
                end
                sync()
              end
              $ 829 "MoveJ"
              $ 830 "Zona_der1" "breakAfter"
              movej(get_inverse_kin(Zona_der1_p, qnear=Zona_der1_q), a=1.3962634015954636, v=1.0471975511965976)
              $ 831 "Posicion_Cero" "breakAfter"
              movej(get_inverse_kin(Posicion_Cero_p, qnear=Posicion_Cero_q), a=1.3962634015954636, v=1.0471975511965976)
              $ 832 "Call Quitar_Broca_Chida"
              Quitar_Broca_Chida()
              $ 833 "Set carrusel_home=Encender"
              modbus_set_output_signal("carrusel_home", True)
              $ 834 "Wait: 1.0"
              sleep(1.0)
              $ 835 "Set carrusel_home=Apagar"
              modbus_set_output_signal("carrusel_home", False)
              $ 836 "Set mensaje_mw10=120"
              modbus_set_output_register("mensaje_mw10", 120)
              $ 837 "Wait Continuar_M30=HI"
              while (modbus_get_signal_status("Continuar_M30") == False):
                sync()
              end
              $ 838 "Wait: 1.0"
              sleep(1.0)
              $ 839 "Set mensaje_mw10=100"
              modbus_set_output_register("mensaje_mw10", 100)
              $ 840 "Wait Continuar_M30=HI"
              while (modbus_get_signal_status("Continuar_M30") == False):
                sync()
              end
              $ 841 "Wait: 1.0"
              sleep(1.0)
              $ 842 "MoveJ"
              $ 843 "Traslacion_der" "breakAfter"
              movej(get_inverse_kin(Traslacion_der_p, qnear=Traslacion_der_q), a=1.3962634015954636, v=1.0471975511965976)
            end
          end
          $ 844 "barrenoActual≔barrenoActual+1"
          global barrenoActual=barrenoActual+1
        end
        $ 845 "Set pos1_term_m611=Encender"
        modbus_set_output_signal("pos1_term_m611", True)
        $ 846 "Wait: 1.0"
        sleep(1.0)
        $ 847 "Set pos1_term_m611=Apagar"
        modbus_set_output_signal("pos1_term_m611", False)
      else:
        $ 848 "ElseIf pos_sig_der≟1"
        if (modbus_get_signal_status("pos_sig_der") == 1):
          $ 849 "Arranque"
          $ 850 "Set mensaje_mw10=15"
          modbus_set_output_register("mensaje_mw10", 15)
          $ 851 "Wait Continuar_M30=HI"
          while (modbus_get_signal_status("Continuar_M30") == False):
            sync()
          end
          $ 852 "Wait: 1.0"
          sleep(1.0)
          $ 853 "MoveJ"
          $ 854 "Off_derecha" "breakAfter"
          movej(get_inverse_kin(Off_derecha_p, qnear=Off_derecha_q), a=1.3962634015954636, v=1.0471975511965976)
          $ 855 "Set postrnas_m187=Encender"
          modbus_set_output_signal("postrnas_m187", True)
          $ 856 "Wait: 1.0"
          sleep(1.0)
          $ 857 "Set Home_M20=Encender"
          modbus_set_output_signal("Home_M20", True)
          $ 858 "Wait: 1.0"
          sleep(1.0)
          $ 859 "Set postrnas_m187=Apagar"
          modbus_set_output_signal("postrnas_m187", False)
          $ 860 "Set Home_M20=Apagar"
          modbus_set_output_signal("Home_M20", False)
          $ 861 "Set mensaje_mw10=20"
          modbus_set_output_register("mensaje_mw10", 20)
          $ 862 "Wait Continuar_M30=HI"
          while (modbus_get_signal_status("Continuar_M30") == False):
            sync()
          end
          $ 863 "Wait: 1.0"
          sleep(1.0)
          $ 864 "Traslacion"
          $ 865 "Set mensaje_mw10=25"
          modbus_set_output_register("mensaje_mw10", 25)
          $ 866 "Wait Continuar_M30=HI"
          while (modbus_get_signal_status("Continuar_M30") == False):
            sync()
          end
          $ 867 "Wait: 1.0"
          sleep(1.0)
          $ 868 "MoveJ"
          $ 869 "Waypoint_8" "breakAfter"
          movej(get_inverse_kin(Waypoint_8_p, qnear=Waypoint_8_q), a=1.3962634015954636, v=1.0471975511965976)
          $ 870 "Traslacion_der" "breakAfter"
          movej(get_inverse_kin(Traslacion_der_p, qnear=Traslacion_der_q), a=1.3962634015954636, v=1.0471975511965976)
          $ 871 "Set mensaje_mw10=105"
          modbus_set_output_register("mensaje_mw10", 105)
          $ 872 "Wait Continuar_M30=HI"
          while (modbus_get_signal_status("Continuar_M30") == False):
            sync()
          end
          $ 873 "Wait: 1.0"
          sleep(1.0)
          $ 874 "Set mensaje_mw10=145"
          modbus_set_output_register("mensaje_mw10", 145)
          $ 875 "Wait Continuar_M30=HI"
          while (modbus_get_signal_status("Continuar_M30") == False):
            sync()
          end
          $ 876 "Wait: 1.0"
          sleep(1.0)
          $ 877 "Set postrnas_m187=Encender"
          modbus_set_output_signal("postrnas_m187", True)
          $ 878 "Wait: 1.0"
          sleep(1.0)
          $ 879 "Set pos2_der_mw698=Encender"
          modbus_set_output_signal("pos2_der_mw698", True)
          $ 880 "Wait: 1.0"
          sleep(1.0)
          $ 881 "Set pos2_der_mw698=Apagar"
          modbus_set_output_signal("pos2_der_mw698", False)
          $ 882 "Set postrnas_m187=Apagar"
          modbus_set_output_signal("postrnas_m187", False)
          $ 883 "Wait: 10.0"
          sleep(10.0)
          $ 884 "Brocas"
          $ 885 "Set carrusel_home=Encender"
          modbus_set_output_signal("carrusel_home", True)
          $ 886 "Wait: 1.0"
          sleep(1.0)
          $ 887 "Set carrusel_home=Apagar"
          modbus_set_output_signal("carrusel_home", False)
          $ 888 "Set mensaje_mw10=40"
          modbus_set_output_register("mensaje_mw10", 40)
          $ 889 "Wait Continuar_M30=HI"
          while (modbus_get_signal_status("Continuar_M30") == False):
            sync()
          end
          $ 890 "Wait: 1.0"
          sleep(1.0)
          $ 891 "Set carrusel_home=Encender"
          modbus_set_output_signal("carrusel_home", True)
          $ 892 "Wait: 1.0"
          sleep(1.0)
          $ 893 "Set carrusel_home=Apagar"
          modbus_set_output_signal("carrusel_home", False)
          $ 894 "Set mensaje_mw10=45"
          modbus_set_output_register("mensaje_mw10", 45)
          $ 895 "Wait Continuar_M30=HI"
          while (modbus_get_signal_status("Continuar_M30") == False):
            sync()
          end
          $ 896 "Wait: 1.0"
          sleep(1.0)
          $ 897 "Call Poner_Broca"
          Poner_Broca()
          $ 898 "Offsets factor"
          $ 900 "L1B1x≔(((0.09525254)/(0.09525))*(0.09525254))*(1)"
          global L1B1x=(((0.09525254)/(0.09525))*(0.09525254))*(1)
          $ 901 "L1B1y≔(((-0.012)/(-0.0127))*(-0.012))*(1)"
          global L1B1y=(((-0.012)/(-0.0127))*(-0.012))*(1)
          $ 902 "L1B2x≔(((0.74)/(0.75565))*(0.74))*(1.0003)"
          global L1B2x=(((0.74)/(0.75565))*(0.74))*(1.0003)
          $ 903 "L1B2y≔(((-0.00986)/(-0.0127))*(-0.00986))*(1.0086956521739)"
          global L1B2y=(((-0.00986)/(-0.0127))*(-0.00986))*(1.0086956521739)
          $ 904 "L2B1x≔((0.09513062)/(0.09525))*(0.09525)"
          global L2B1x=((0.09513062)/(0.09525))*(0.09525)
          $ 905 "L2B1y≔((0.39369238)/(0.3937))*(0.39369238)"
          global L2B1y=((0.39369238)/(0.3937))*(0.39369238)
          $ 906 "L2B2x≔((0.75565508)/(0.75565))*(0.75565508)"
          global L2B2x=((0.75565508)/(0.75565))*(0.75565508)
          $ 907 "L2B2y≔((0.39290032)/(0.3937))*(0.39290032)"
          global L2B2y=((0.39290032)/(0.3937))*(0.39290032)
          $ 908 "Calibracion"
          $ 909 "Set mensaje_mw10=50"
          modbus_set_output_register("mensaje_mw10", 50)
          $ 910 "Wait Continuar_M30=HI"
          while (modbus_get_signal_status("Continuar_M30") == False):
            sync()
          end
          $ 911 "Wait: 1.0"
          sleep(1.0)
          $ 912 "MoveJ"
          $ 913 "Posicion_Cero" "breakAfter"
          movej(get_inverse_kin(Posicion_Cero_p, qnear=Posicion_Cero_q), a=1.3962634015954636, v=1.0471975511965976)
          $ 914 "Zona_der1" "breakAfter"
          movej(get_inverse_kin(Zona_der1_p, qnear=Zona_der1_q), a=1.3962634015954636, v=1.0471975511965976)
          $ 915 "broca≔1645"
          global broca=1645
          $ 916 "Set mensaje_mw10=125"
          modbus_set_output_register("mensaje_mw10", 125)
          $ 917 "Wait Continuar_M30=HI"
          while (modbus_get_signal_status("Continuar_M30") == False):
            sync()
          end
          $ 918 "Wait: 1.0"
          sleep(1.0)
          $ 919 "Set mensaje_mw10=130"
          modbus_set_output_register("mensaje_mw10", 130)
          $ 920 "Wait Continuar_M30=HI"
          while (modbus_get_signal_status("Continuar_M30") == False):
            sync()
          end
          $ 921 "Wait: 1.0"
          sleep(1.0)
          $ 922 "Call Calibracion"
          Calibracion()
          $ 923 "GoNoGo"
          $ 924 "Set mensaje_mw10=55"
          modbus_set_output_register("mensaje_mw10", 55)
          $ 925 "Wait Continuar_M30=HI"
          while (modbus_get_signal_status("Continuar_M30") == False):
            sync()
          end
          $ 926 "Wait: 1.0"
          sleep(1.0)
          $ 927 "Set mensaje_mw10=60"
          modbus_set_output_register("mensaje_mw10", 60)
          $ 928 "Wait Continuar_M30=HI"
          while (modbus_get_signal_status("Continuar_M30") == False):
            sync()
          end
          $ 929 "Wait: 1.0"
          sleep(1.0)
          $ 930 "Linea1_Buje1"
          $ 931 "Xfin≔(((L1B1x)*Xp)-(Xd)-((L1B1y)*(1/m2)))*(-1)"
          global Xfin=(((L1B1x)*Xp)-(Xd)-((L1B1y)*(1/m2)))*(-1)
          $ 932 "Yfin≔(((L1B1y)*Yp)-(Yd)+((L1B1x)*m1))*(-1)"
          global Yfin=(((L1B1y)*Yp)-(Yd)+((L1B1x)*m1))*(-1)
          $ 933 "rotaciones≔get_actual_tcp_pose()"
          global rotaciones= get_actual_tcp_pose ()
          $ 934 "var_3≔rotaciones[3]"
          global var_3=rotaciones[3]
          $ 935 "var_4≔rotaciones[4]"
          global var_4=rotaciones[4]
          $ 936 "var_5≔rotaciones[5]"
          global var_5=rotaciones[5]
          $ 937 "If broca≟1645"
          if (broca == 1645):
            $ 938 "PosFinal≔p[Xfin+0.00208915,Yfin+0.00208915,0.1,var_3,var_4,var_5]"
            global PosFinal=p[Xfin+0.00208915,Yfin+0.00208915,0.1,var_3,var_4,var_5]
          else:
            $ 939 "ElseIf broca≟1935"
            if (broca == 1935):
              $ 940 "PosFinal≔p[Xfin+0.00245745,Yfin+0.00245745,0.1,var_3,var_4,var_5]"
              global PosFinal=p[Xfin+0.00245745,Yfin+0.00245745,0.1,var_3,var_4,var_5]
            else:
              $ 941 "ElseIf broca≟217"
              if (broca == 217):
                $ 942 "PosFinal≔p[Xfin+0.0027559,Yfin+0.0027559,0.1,var_3,var_4,var_5]"
                global PosFinal=p[Xfin+0.0027559,Yfin+0.0027559,0.1,var_3,var_4,var_5]
              end
            end
          end
          $ 943 "Buje_Final≔PosFinal"
          global Buje_Final=PosFinal
          $ 944 "MoveJ"
          $ 945 "Buje_Final" "breakAfter"
          movej(Buje_Final, a=1.3962634015954636, v=1.0471975511965976)
          $ 946 "Wait: 1.0"
          sleep(1.0)
          $ 947 "Alturas"
          $ 948 "If P1h[2]<P2h[2]"
          if (P1h[2]<P2h[2]):
            $ 949 "tcp≔get_actual_tcp_pose()"
            global tcp= get_actual_tcp_pose ()
            $ 950 "offset_altura≔p[tcp[0],tcp[1],((alta-0.0095)-(altura/1000)),tcp[3],tcp[4],tcp[5]]"
            global offset_altura=p[tcp[0],tcp[1],((alta-0.0095)-(altura/1000)),tcp[3],tcp[4],tcp[5]]
            $ 951 "MoveL"
            $ 952 "offset_altura" "breakAfter"
            movel(offset_altura, a=0.04, v=0.03)
          else:
            $ 953 "Else" "noBreak"
            $ 954 "tcp≔get_actual_tcp_pose()"
            global tcp= get_actual_tcp_pose ()
            $ 955 "offset_altura≔p[tcp[0],tcp[1],((alta-0.0095)),tcp[3],tcp[4],tcp[5]]"
            global offset_altura=p[tcp[0],tcp[1],((alta-0.0095)),tcp[3],tcp[4],tcp[5]]
            $ 956 "MoveL"
            $ 957 "offset_altura" "breakAfter"
            movel(offset_altura, a=0.04, v=0.03)
          end
          $ 958 "MoveL"
          $ 959 "Freemove"
          $ 960 "Wait: 2.0"
          sleep(2.0)
          $ 961 "freedrive_mode()"
          freedrive_mode()
          $ 962 "Wait: 2.5"
          sleep(2.5)
          $ 963 "end_freedrive_mode()"
          end_freedrive_mode()
          $ 964 "var_11≔get_actual_tcp_pose()"
          global var_11= get_actual_tcp_pose ()
          $ 965 "var_11≔p[var_11[0]*1000,var_11[1]*1000,420,420,420,420]"
          global var_11=p[var_11[0]*1000,var_11[1]*1000,420,420,420,420]
          $ 966 "var_11≔get_actual_tcp_pose()"
          global var_11= get_actual_tcp_pose ()
          $ 967 "var_11≔p[var_11[0],var_11[1],0.1,var_11[3],var_11[4],var_11[5]]"
          global var_11=p[var_11[0],var_11[1],0.1,var_11[3],var_11[4],var_11[5]]
          $ 968 "Direction: Base Z+"
          global move_thread_flag_968=0
          thread move_thread_968():
            enter_critical
            move_thread_flag_968 = 1
            local towardsPos=calculate_point_to_move_towards(p[0.0,0.0,0.0,0.0,0.0,0.0], [0.0,0.0,1.0], 0.15)
            movel(towardsPos, a=0.08, v=0.06)
            move_thread_flag_968 = 2
            exit_critical
          end
          move_thread_flag_968 = 0
          move_thread_han_968 = run move_thread_968()
          while (True):
            sleep(1.0E-10)
            if (move_thread_flag_968 > 1):
              join move_thread_han_968
              $ 969 "Until (distance)"
              break
            end
            sync()
          end
          $ 970 "Direction: Base X-"
          global move_thread_flag_970=0
          thread move_thread_970():
            enter_critical
            move_thread_flag_970 = 1
            local towardsPos=calculate_point_to_move_towards(p[0.0,0.0,0.0,0.0,0.0,0.0], [-1.0,0.0,0.0], 0.42)
            movel(towardsPos, a=0.08, v=0.06)
            move_thread_flag_970 = 2
            exit_critical
          end
          move_thread_flag_970 = 0
          move_thread_han_970 = run move_thread_970()
          while (True):
            sleep(1.0E-10)
            if (move_thread_flag_970 > 1):
              join move_thread_han_970
              $ 971 "Until (distance)"
              break
            end
            sync()
          end
          $ 972 "L1B1≔var_11"
          global L1B1=var_11
          $ 973 "Linea1_Buje2"
          $ 974 "Xfin≔(((L1B2x)*Xp)-(Xd)-((L1B2y)*(1/m2)))*(-1)"
          global Xfin=(((L1B2x)*Xp)-(Xd)-((L1B2y)*(1/m2)))*(-1)
          $ 975 "Yfin≔(((L1B2y)*Yp)-(Yd)+((L1B2x)*m1))*(-1)"
          global Yfin=(((L1B2y)*Yp)-(Yd)+((L1B2x)*m1))*(-1)
          $ 976 "rotaciones≔get_actual_tcp_pose()"
          global rotaciones= get_actual_tcp_pose ()
          $ 977 "var_3≔rotaciones[3]"
          global var_3=rotaciones[3]
          $ 978 "var_4≔rotaciones[4]"
          global var_4=rotaciones[4]
          $ 979 "var_5≔rotaciones[5]"
          global var_5=rotaciones[5]
          $ 980 "If broca≟1645"
          if (broca == 1645):
            $ 981 "PosFinal≔p[Xfin+0.00208915,Yfin+0.00208915,0.1,var_3,var_4,var_5]"
            global PosFinal=p[Xfin+0.00208915,Yfin+0.00208915,0.1,var_3,var_4,var_5]
          else:
            $ 982 "ElseIf broca≟1935"
            if (broca == 1935):
              $ 983 "PosFinal≔p[Xfin+0.00245745,Yfin+0.00245745,0.1,var_3,var_4,var_5]"
              global PosFinal=p[Xfin+0.00245745,Yfin+0.00245745,0.1,var_3,var_4,var_5]
            else:
              $ 984 "ElseIf broca≟217"
              if (broca == 217):
                $ 985 "PosFinal≔p[Xfin+0.0027559,Yfin+0.0027559,0.1,var_3,var_4,var_5]"
                global PosFinal=p[Xfin+0.0027559,Yfin+0.0027559,0.1,var_3,var_4,var_5]
              end
            end
          end
          $ 986 "Buje_Final≔PosFinal"
          global Buje_Final=PosFinal
          $ 987 "MoveJ"
          $ 988 "Buje_Final" "breakAfter"
          movej(Buje_Final, a=1.3962634015954636, v=1.0471975511965976)
          $ 989 "Wait: 1.0"
          sleep(1.0)
          $ 990 "Alturas"
          $ 991 "If P1h[2]<P2h[2]"
          if (P1h[2]<P2h[2]):
            $ 992 "tcp≔get_actual_tcp_pose()"
            global tcp= get_actual_tcp_pose ()
            $ 993 "offset_altura≔p[tcp[0],tcp[1],((alta-0.0095)),tcp[3],tcp[4],tcp[5]]"
            global offset_altura=p[tcp[0],tcp[1],((alta-0.0095)),tcp[3],tcp[4],tcp[5]]
            $ 994 "MoveL"
            $ 995 "offset_altura" "breakAfter"
            movel(offset_altura, a=0.04, v=0.03)
          else:
            $ 996 "Else" "noBreak"
            $ 997 "tcp≔get_actual_tcp_pose()"
            global tcp= get_actual_tcp_pose ()
            $ 998 "offset_altura≔p[tcp[0],tcp[1],((alta-0.0095)-(altura/1000)),tcp[3],tcp[4],tcp[5]]"
            global offset_altura=p[tcp[0],tcp[1],((alta-0.0095)-(altura/1000)),tcp[3],tcp[4],tcp[5]]
            $ 999 "MoveL"
            $ 1000 "offset_altura" "breakAfter"
            movel(offset_altura, a=0.04, v=0.03)
          end
          $ 1001 "MoveL"
          $ 1002 "Freemove"
          $ 1003 "Wait: 2.0"
          sleep(2.0)
          $ 1004 "freedrive_mode()"
          freedrive_mode()
          $ 1005 "Wait: 2.5"
          sleep(2.5)
          $ 1006 "end_freedrive_mode()"
          end_freedrive_mode()
          $ 1007 "var_11≔get_actual_tcp_pose()"
          global var_11= get_actual_tcp_pose ()
          $ 1008 "var_11≔p[var_11[0]*1000,var_11[1]*1000,420,420,420,420]"
          global var_11=p[var_11[0]*1000,var_11[1]*1000,420,420,420,420]
          $ 1009 "var_11≔get_actual_tcp_pose()"
          global var_11= get_actual_tcp_pose ()
          $ 1010 "var_11≔p[var_11[0],var_11[1],0.1,var_11[3],var_11[4],var_11[5]]"
          global var_11=p[var_11[0],var_11[1],0.1,var_11[3],var_11[4],var_11[5]]
          $ 1011 "Direction: Base Z+"
          global move_thread_flag_1011=0
          thread move_thread_1011():
            enter_critical
            move_thread_flag_1011 = 1
            local towardsPos=calculate_point_to_move_towards(p[0.0,0.0,0.0,0.0,0.0,0.0], [0.0,0.0,1.0], 0.15)
            movel(towardsPos, a=0.08, v=0.06)
            move_thread_flag_1011 = 2
            exit_critical
          end
          move_thread_flag_1011 = 0
          move_thread_han_1011 = run move_thread_1011()
          while (True):
            sleep(1.0E-10)
            if (move_thread_flag_1011 > 1):
              join move_thread_han_1011
              $ 1012 "Until (distance)"
              break
            end
            sync()
          end
          $ 1013 "L1B2≔var_11"
          global L1B2=var_11
          $ 1014 "Linea2_Buje2"
          $ 1015 "Xfin≔(((L2B2x)*Xp)-(Xd)-((L2B2y)*(1/m2)))*(-1)"
          global Xfin=(((L2B2x)*Xp)-(Xd)-((L2B2y)*(1/m2)))*(-1)
          $ 1016 "Yfin≔(((L2B2y)*Yp)-(Yd)+((L2B2x)*m1))*(-1)"
          global Yfin=(((L2B2y)*Yp)-(Yd)+((L2B2x)*m1))*(-1)
          $ 1017 "rotaciones≔get_actual_tcp_pose()"
          global rotaciones= get_actual_tcp_pose ()
          $ 1018 "var_3≔rotaciones[3]"
          global var_3=rotaciones[3]
          $ 1019 "var_4≔rotaciones[4]"
          global var_4=rotaciones[4]
          $ 1020 "var_5≔rotaciones[5]"
          global var_5=rotaciones[5]
          $ 1021 "If broca≟1645"
          if (broca == 1645):
            $ 1022 "PosFinal≔p[Xfin+0.00208915,Yfin+0.00208915,0.1,var_3,var_4,var_5]"
            global PosFinal=p[Xfin+0.00208915,Yfin+0.00208915,0.1,var_3,var_4,var_5]
          else:
            $ 1023 "ElseIf broca≟1935"
            if (broca == 1935):
              $ 1024 "PosFinal≔p[Xfin+0.00245745,Yfin+0.00245745,0.1,var_3,var_4,var_5]"
              global PosFinal=p[Xfin+0.00245745,Yfin+0.00245745,0.1,var_3,var_4,var_5]
            else:
              $ 1025 "ElseIf broca≟217"
              if (broca == 217):
                $ 1026 "PosFinal≔p[Xfin+0.0027559,Yfin+0.0027559,0.1,var_3,var_4,var_5]"
                global PosFinal=p[Xfin+0.0027559,Yfin+0.0027559,0.1,var_3,var_4,var_5]
              end
            end
          end
          $ 1027 "Buje_Final≔PosFinal"
          global Buje_Final=PosFinal
          $ 1028 "MoveJ"
          $ 1029 "Buje_Final" "breakAfter"
          movej(Buje_Final, a=1.3962634015954636, v=1.0471975511965976)
          $ 1030 "Wait: 1.0"
          sleep(1.0)
          $ 1031 "Alturas"
          $ 1032 "If P1h[2]<P2h[2]"
          if (P1h[2]<P2h[2]):
            $ 1033 "tcp≔get_actual_tcp_pose()"
            global tcp= get_actual_tcp_pose ()
            $ 1034 "offset_altura≔p[tcp[0],tcp[1],((alta-0.0095)),tcp[3],tcp[4],tcp[5]]"
            global offset_altura=p[tcp[0],tcp[1],((alta-0.0095)),tcp[3],tcp[4],tcp[5]]
            $ 1035 "MoveL"
            $ 1036 "offset_altura" "breakAfter"
            movel(offset_altura, a=0.04, v=0.03)
          else:
            $ 1037 "Else" "noBreak"
            $ 1038 "tcp≔get_actual_tcp_pose()"
            global tcp= get_actual_tcp_pose ()
            $ 1039 "offset_altura≔p[tcp[0],tcp[1],((alta-0.0095)-(altura/1000)),tcp[3],tcp[4],tcp[5]]"
            global offset_altura=p[tcp[0],tcp[1],((alta-0.0095)-(altura/1000)),tcp[3],tcp[4],tcp[5]]
            $ 1040 "MoveL"
            $ 1041 "offset_altura" "breakAfter"
            movel(offset_altura, a=0.04, v=0.03)
          end
          $ 1042 "MoveL"
          $ 1043 "Freemove"
          $ 1044 "Wait: 2.0"
          sleep(2.0)
          $ 1045 "freedrive_mode()"
          freedrive_mode()
          $ 1046 "Wait: 2.5"
          sleep(2.5)
          $ 1047 "end_freedrive_mode()"
          end_freedrive_mode()
          $ 1048 "var_11≔get_actual_tcp_pose()"
          global var_11= get_actual_tcp_pose ()
          $ 1049 "var_11≔p[var_11[0]*1000,var_11[1]*1000,420,420,420,420]"
          global var_11=p[var_11[0]*1000,var_11[1]*1000,420,420,420,420]
          $ 1050 "var_11≔get_actual_tcp_pose()"
          global var_11= get_actual_tcp_pose ()
          $ 1051 "var_11≔p[var_11[0],var_11[1],0.1,var_11[3],var_11[4],var_11[5]]"
          global var_11=p[var_11[0],var_11[1],0.1,var_11[3],var_11[4],var_11[5]]
          $ 1052 "Direction: Base Z+"
          global move_thread_flag_1052=0
          thread move_thread_1052():
            enter_critical
            move_thread_flag_1052 = 1
            local towardsPos=calculate_point_to_move_towards(p[0.0,0.0,0.0,0.0,0.0,0.0], [0.0,0.0,1.0], 0.15)
            movel(towardsPos, a=0.08, v=0.06)
            move_thread_flag_1052 = 2
            exit_critical
          end
          move_thread_flag_1052 = 0
          move_thread_han_1052 = run move_thread_1052()
          while (True):
            sleep(1.0E-10)
            if (move_thread_flag_1052 > 1):
              join move_thread_han_1052
              $ 1053 "Until (distance)"
              break
            end
            sync()
          end
          $ 1054 "L2B2≔var_11"
          global L2B2=var_11
          $ 1055 "Linea2_Buje1"
          $ 1056 "Xfin≔(((L2B1x)*Xp)-(Xd)-((L2B1y)*(1/m2)))*(-1)"
          global Xfin=(((L2B1x)*Xp)-(Xd)-((L2B1y)*(1/m2)))*(-1)
          $ 1057 "Yfin≔(((L2B1y)*Yp)-(Yd)+((L2B1x)*m1))*(-1)"
          global Yfin=(((L2B1y)*Yp)-(Yd)+((L2B1x)*m1))*(-1)
          $ 1058 "rotaciones≔get_actual_tcp_pose()"
          global rotaciones= get_actual_tcp_pose ()
          $ 1059 "var_3≔rotaciones[3]"
          global var_3=rotaciones[3]
          $ 1060 "var_4≔rotaciones[4]"
          global var_4=rotaciones[4]
          $ 1061 "var_5≔rotaciones[5]"
          global var_5=rotaciones[5]
          $ 1062 "If broca≟1645"
          if (broca == 1645):
            $ 1063 "PosFinal≔p[Xfin+0.00208915,Yfin+0.00208915,0.1,var_3,var_4,var_5]"
            global PosFinal=p[Xfin+0.00208915,Yfin+0.00208915,0.1,var_3,var_4,var_5]
          else:
            $ 1064 "ElseIf broca≟1935"
            if (broca == 1935):
              $ 1065 "PosFinal≔p[Xfin+0.00245745,Yfin+0.00245745,0.1,var_3,var_4,var_5]"
              global PosFinal=p[Xfin+0.00245745,Yfin+0.00245745,0.1,var_3,var_4,var_5]
            else:
              $ 1066 "ElseIf broca≟217"
              if (broca == 217):
                $ 1067 "PosFinal≔p[Xfin+0.0027559,Yfin+0.0027559,0.1,var_3,var_4,var_5]"
                global PosFinal=p[Xfin+0.0027559,Yfin+0.0027559,0.1,var_3,var_4,var_5]
              end
            end
          end
          $ 1068 "Buje_Final≔PosFinal"
          global Buje_Final=PosFinal
          $ 1069 "MoveJ"
          $ 1070 "Buje_Final" "breakAfter"
          movej(Buje_Final, a=1.3962634015954636, v=1.0471975511965976)
          $ 1071 "Wait: 1.0"
          sleep(1.0)
          $ 1072 "Alturas"
          $ 1073 "If P1h[2]<P2h[2]"
          if (P1h[2]<P2h[2]):
            $ 1074 "tcp≔get_actual_tcp_pose()"
            global tcp= get_actual_tcp_pose ()
            $ 1075 "offset_altura≔p[tcp[0],tcp[1],((alta-0.0095)-(altura/1000)),tcp[3],tcp[4],tcp[5]]"
            global offset_altura=p[tcp[0],tcp[1],((alta-0.0095)-(altura/1000)),tcp[3],tcp[4],tcp[5]]
            $ 1076 "MoveL"
            $ 1077 "offset_altura" "breakAfter"
            movel(offset_altura, a=0.04, v=0.03)
          else:
            $ 1078 "Else" "noBreak"
            $ 1079 "tcp≔get_actual_tcp_pose()"
            global tcp= get_actual_tcp_pose ()
            $ 1080 "offset_altura≔p[tcp[0],tcp[1],((alta-0.0095)),tcp[3],tcp[4],tcp[5]]"
            global offset_altura=p[tcp[0],tcp[1],((alta-0.0095)),tcp[3],tcp[4],tcp[5]]
            $ 1081 "MoveL"
            $ 1082 "offset_altura" "breakAfter"
            movel(offset_altura, a=0.04, v=0.03)
          end
          $ 1083 "MoveL"
          $ 1084 "Freemove"
          $ 1085 "Wait: 2.0"
          sleep(2.0)
          $ 1086 "freedrive_mode()"
          freedrive_mode()
          $ 1087 "Wait: 2.5"
          sleep(2.5)
          $ 1088 "end_freedrive_mode()"
          end_freedrive_mode()
          $ 1089 "var_11≔get_actual_tcp_pose()"
          global var_11= get_actual_tcp_pose ()
          $ 1090 "var_11≔p[var_11[0]*1000,var_11[1]*1000,420,420,420,420]"
          global var_11=p[var_11[0]*1000,var_11[1]*1000,420,420,420,420]
          $ 1091 "var_11≔get_actual_tcp_pose()"
          global var_11= get_actual_tcp_pose ()
          $ 1092 "var_11≔p[var_11[0],var_11[1],0.1,var_11[3],var_11[4],var_11[5]]"
          global var_11=p[var_11[0],var_11[1],0.1,var_11[3],var_11[4],var_11[5]]
          $ 1093 "Direction: Base Z+"
          global move_thread_flag_1093=0
          thread move_thread_1093():
            enter_critical
            move_thread_flag_1093 = 1
            local towardsPos=calculate_point_to_move_towards(p[0.0,0.0,0.0,0.0,0.0,0.0], [0.0,0.0,1.0], 0.15)
            movel(towardsPos, a=0.08, v=0.06)
            move_thread_flag_1093 = 2
            exit_critical
          end
          move_thread_flag_1093 = 0
          move_thread_han_1093 = run move_thread_1093()
          while (True):
            sleep(1.0E-10)
            if (move_thread_flag_1093 > 1):
              join move_thread_han_1093
              $ 1094 "Until (distance)"
              break
            end
            sync()
          end
          $ 1095 "L2B1≔var_11"
          global L2B1=var_11
          $ 1096 "MoveJ"
          $ 1097 "Zona_der1" "breakAfter"
          movej(get_inverse_kin(Zona_der1_p, qnear=Zona_der1_q), a=1.3962634015954636, v=1.0471975511965976)
          $ 1113 "Colocar broca"
          $ 1114 "Call Quitar_Broca_Chida"
          Quitar_Broca_Chida()
          $ 1115 "Call Poner_Broca"
          Poner_Broca()
          $ 1116 "Barrenado"
          $ 1117 "Set mensaje_mw10=65"
          modbus_set_output_register("mensaje_mw10", 65)
          $ 1118 "Wait Continuar_M30=HI"
          while (modbus_get_signal_status("Continuar_M30") == False):
            sync()
          end
          $ 1119 "Wait: 1.0"
          sleep(1.0)
          $ 1120 "Set mensaje_mw10=150"
          modbus_set_output_register("mensaje_mw10", 150)
          $ 1121 "Wait: 1.0"
          sleep(1.0)
          $ 1122 "Linea 1 a 1645"
          $ 1123 "broca≔1645"
          global broca=1645
          $ 1124 "Buje_inicial"
          $ 1125 "Buje_Inicial≔L1B2"
          global Buje_Inicial=L1B2
          $ 1126 "Buje_final"
          $ 1127 "Buje_Final≔L1B1"
          global Buje_Final=L1B1
          $ 1128 "barrenosTotales≔27"
          global barrenosTotales=27
          $ 1129 "barrenoActual≔1"
          global barrenoActual=1
          $ 1130 "Loop barrenoActual≤barrenosTotales"
          while (barrenoActual <= barrenosTotales):
            $ 1131 "MoveL"
            $ 1132 "bajada_broca≔p[0,0,0.006,0,0,0]"
            global bajada_broca=p[0,0,0.006,0,0,0]
            $ 1133 "internos≔interpolate_pose(Buje_Inicial, Buje_Final, ((barrenoActual)-1)/((barrenosTotales)-1))"
            global internos= interpolate_pose (Buje_Inicial, Buje_Final, ((barrenoActual)-1)/((barrenosTotales)-1))
            $ 1134 "If barrenoActual≟1 or barrenoActual≟3 or barrenoActual≟5 or barrenoActual≟7 or barrenoActual≟9 or barrenoActual≟11 or barrenoActual≟13 or barrenoActual≟15 or barrenoActual≟17 or barrenoActual≟19 or barrenoActual≟21 or barrenoActual≟23 or barrenoActual≟25 or barrenoActual≟27"
            if (barrenoActual == 1  or  barrenoActual == 3  or  barrenoActual == 5  or  barrenoActual == 7  or  barrenoActual == 9  or  barrenoActual == 11  or  barrenoActual == 13  or  barrenoActual == 15  or  barrenoActual == 17  or  barrenoActual == 19  or  barrenoActual == 21  or  barrenoActual == 23  or  barrenoActual == 25  or  barrenoActual == 27):
              $ 1135 "Set mensaje_mw10=200"
              modbus_set_output_register("mensaje_mw10", 200)
              $ 1136 "Wait Continuar_M30=HI"
              while (modbus_get_signal_status("Continuar_M30") == False):
                sync()
              end
              $ 1137 "Wait: 1.0"
              sleep(1.0)
              $ 1138 "Set mensaje_mw10=150"
              modbus_set_output_register("mensaje_mw10", 150)
              $ 1139 "Wait: 1.0"
              sleep(1.0)
            end
            $ 1140 "MoveJ"
            $ 1141 "internos" "breakAfter"
            movej(internos, a=0.6981317007977318, v=0.5235987755982988)
            $ 1142 "Wait: 2.0"
            sleep(2.0)
            $ 1143 "Alturas"
            $ 1144 "If P1h[2]<P2h[2]"
            if (P1h[2]<P2h[2]):
              $ 1145 "acomodo≔(altura/(barrenosTotales-1))*(barrenoActual-1)"
              global acomodo=(altura/(barrenosTotales-1))*(barrenoActual-1)
              $ 1146 "tcp≔get_actual_tcp_pose()"
              global tcp= get_actual_tcp_pose ()
              $ 1147 "offset_altura≔p[tcp[0],tcp[1],((alta-0.0095)-(acomodo/1000)),tcp[3],tcp[4],tcp[5]]"
              global offset_altura=p[tcp[0],tcp[1],((alta-0.0095)-(acomodo/1000)),tcp[3],tcp[4],tcp[5]]
              $ 1148 "MoveL"
              $ 1149 "offset_altura" "breakAfter"
              movel(offset_altura, a=0.04, v=0.03)
            else:
              $ 1150 "Else" "noBreak"
              $ 1151 "acomodo≔(altura/(barrenosTotales-1))*(26-(barrenoActual-1))"
              global acomodo=(altura/(barrenosTotales-1))*(26-(barrenoActual-1))
              $ 1152 "tcp≔get_actual_tcp_pose()"
              global tcp= get_actual_tcp_pose ()
              $ 1153 "offset_altura≔p[tcp[0],tcp[1],((alta-0.0095)-(acomodo/1000)),tcp[3],tcp[4],tcp[5]]"
              global offset_altura=p[tcp[0],tcp[1],((alta-0.0095)-(acomodo/1000)),tcp[3],tcp[4],tcp[5]]
              $ 1154 "MoveL"
              $ 1155 "offset_altura" "breakAfter"
              movel(offset_altura, a=0.04, v=0.03)
            end
            $ 1156 "Freemove"
            $ 1157 "Wait: 2.0"
            sleep(2.0)
            $ 1158 "freedrive_mode()"
            freedrive_mode()
            $ 1159 "Wait: 2.5"
            sleep(2.5)
            $ 1160 "end_freedrive_mode()"
            end_freedrive_mode()
            $ 1161 "Wait: 0.3"
            sleep(0.3)
            $ 1162 "Set CO[1]=Encender"
            set_configurable_digital_out(1, True)
            $ 1163 "Wait: 1.0"
            sleep(1.0)
            $ 1164 "Wait: 0.3"
            sleep(0.3)
            $ 1165 "Wait: 0.3"
            sleep(0.3)
            $ 1166 "Wait: 0.3"
            sleep(0.3)
            $ 1167 "Loop 3 times"
            Loop_42 = 0
            while (Loop_42 < 3):
              $ 1168 "Poses_taladrado≔pose_sub(get_actual_tcp_pose(), bajada_broca)"
              global Poses_taladrado= pose_sub ( get_actual_tcp_pose (), bajada_broca)
              $ 1169 "Poses_taladrado" "breakAfter"
              movel(Poses_taladrado, a=0.005, v=0.001)
              $ 1170 "If bajada_broca≟p[0,0,0.018,0,0,0]"
              if (bajada_broca == p[0,0,0.018,0,0,0]):
                $ 1171 "num_barreno≔str_cat('Barreno: ',barrenoActual)"
                global num_barreno=str_cat("Barreno: ",barrenoActual)
                $ 1172 "tcp_actual≔get_actual_tcp_pose()"
                global tcp_actual= get_actual_tcp_pose ()
                $ 1173 "X_actual≔str_cat('     X: ',tcp_actual[0])"
                global X_actual=str_cat("     X: ",tcp_actual[0])
                $ 1174 "Y_actual≔str_cat('     Y: ',tcp_actual[1])"
                global Y_actual=str_cat("     Y: ",tcp_actual[1])
                $ 1175 "pos_barreno≔str_cat(X_actual,Y_actual)"
                global pos_barreno=str_cat(X_actual,Y_actual)
                $ 1176 "textmsg(num_barreno,pos_barreno)"
                textmsg(num_barreno,pos_barreno)
              end
              $ 1177 "Poses_taladrado≔pose_add(get_actual_tcp_pose(), bajada_broca)"
              global Poses_taladrado= pose_add ( get_actual_tcp_pose (), bajada_broca)
              $ 1178 "Poses_taladrado" "breakAfter"
              movel(Poses_taladrado, a=0.01, v=0.01)
              $ 1179 "bajada_broca≔pose_add(bajada_broca, p[0,0,0.006,0,0,0])"
              global bajada_broca= pose_add (bajada_broca, p[0,0,0.006,0,0,0])
              Loop_42 = Loop_42 + 1
            end
            $ 1180 "Direction: Base Z+"
            global move_thread_flag_1180=0
            thread move_thread_1180():
              enter_critical
              move_thread_flag_1180 = 1
              local towardsPos=calculate_point_to_move_towards(p[0.0,0.0,0.0,0.0,0.0,0.0], [0.0,0.0,1.0], 0.05)
              movel(towardsPos, a=0.04, v=0.03)
              move_thread_flag_1180 = 2
              exit_critical
            end
            move_thread_flag_1180 = 0
            move_thread_han_1180 = run move_thread_1180()
            while (True):
              sleep(1.0E-10)
              if (move_thread_flag_1180 > 1):
                join move_thread_han_1180
                $ 1181 "Until (distance)"
                break
              end
              sync()
            end
            $ 1182 "MoveJ"
            $ 1183 "internos" "breakAfter"
            movej(internos, a=0.6981317007977318, v=0.5235987755982988)
            $ 1184 "Wait: 0.3"
            sleep(0.3)
            $ 1185 "Set CO[1]=Apagar"
            set_configurable_digital_out(1, False)
            $ 1186 "Wait: 0.3"
            sleep(0.3)
            $ 1187 "If barrenoActual≟13 or barrenoActual≟27"
            if (barrenoActual == 13  or  barrenoActual == 27):
              $ 1188 "Direction: Base Z+"
              global move_thread_flag_1188=0
              thread move_thread_1188():
                enter_critical
                move_thread_flag_1188 = 1
                local towardsPos=calculate_point_to_move_towards(p[0.0,0.0,0.0,0.0,0.0,0.0], [0.0,0.0,1.0], 0.03)
                movel(towardsPos, a=0.04, v=0.03)
                move_thread_flag_1188 = 2
                exit_critical
              end
              move_thread_flag_1188 = 0
              move_thread_han_1188 = run move_thread_1188()
              while (True):
                sleep(1.0E-10)
                if (move_thread_flag_1188 > 1):
                  join move_thread_han_1188
                  $ 1189 "Until (distance)"
                  break
                end
                sync()
              end
              $ 1190 "MoveJ"
              $ 1191 "Zona_der1" "breakAfter"
              movej(get_inverse_kin(Zona_der1_p, qnear=Zona_der1_q), a=0.6981317007977318, v=0.5235987755982988)
              $ 1192 "Posicion_Cero" "breakAfter"
              movej(get_inverse_kin(Posicion_Cero_p, qnear=Posicion_Cero_q), a=0.6981317007977318, v=0.5235987755982988)
              $ 1193 "Call Quitar_Broca_Chida"
              Quitar_Broca_Chida()
              $ 1194 "If barrenoActual≟13"
              if (barrenoActual == 13):
                $ 1195 "Call Poner_Broca"
                Poner_Broca()
              else:
                $ 1196 "ElseIf barrenoActual≟27"
                if (barrenoActual == 27):
                  $ 1197 "Call Poner_Broca"
                  Poner_Broca()
                end
              end
              $ 1198 "MoveJ"
              $ 1199 "Posicion_Cero" "breakAfter"
              movej(get_inverse_kin(Posicion_Cero_p, qnear=Posicion_Cero_q), a=0.6981317007977318, v=0.5235987755982988)
              $ 1200 "Zona_der1" "breakAfter"
              movej(get_inverse_kin(Zona_der1_p, qnear=Zona_der1_q), a=0.6981317007977318, v=0.5235987755982988)
            end
            $ 1201 "barrenoActual≔barrenoActual+1"
            global barrenoActual=barrenoActual+1
          end
          $ 1202 "Linea 2 a 1645"
          $ 1203 "broca≔1645"
          global broca=1645
          $ 1204 "Buje_inicial"
          $ 1205 "Buje_Inicial≔L2B2"
          global Buje_Inicial=L2B2
          $ 1206 "Buje_final"
          $ 1207 "Buje_Final≔L2B1"
          global Buje_Final=L2B1
          $ 1208 "barrenosTotales≔27"
          global barrenosTotales=27
          $ 1209 "barrenoActual≔1"
          global barrenoActual=1
          $ 1210 "Loop barrenoActual≤barrenosTotales"
          while (barrenoActual <= barrenosTotales):
            $ 1211 "MoveL"
            $ 1212 "bajada_broca≔p[0,0,0.006,0,0,0]"
            global bajada_broca=p[0,0,0.006,0,0,0]
            $ 1213 "internos≔interpolate_pose(Buje_Inicial, Buje_Final, ((barrenoActual)-1)/((barrenosTotales)-1))"
            global internos= interpolate_pose (Buje_Inicial, Buje_Final, ((barrenoActual)-1)/((barrenosTotales)-1))
            $ 1214 "Alturas"
            $ 1215 "If barrenoActual≟1 or barrenoActual≟3 or barrenoActual≟5 or barrenoActual≟7 or barrenoActual≟9 or barrenoActual≟11 or barrenoActual≟13 or barrenoActual≟15 or barrenoActual≟17 or barrenoActual≟19 or barrenoActual≟21 or barrenoActual≟23 or barrenoActual≟25 or barrenoActual≟27"
            if (barrenoActual == 1  or  barrenoActual == 3  or  barrenoActual == 5  or  barrenoActual == 7  or  barrenoActual == 9  or  barrenoActual == 11  or  barrenoActual == 13  or  barrenoActual == 15  or  barrenoActual == 17  or  barrenoActual == 19  or  barrenoActual == 21  or  barrenoActual == 23  or  barrenoActual == 25  or  barrenoActual == 27):
              $ 1216 "Set mensaje_mw10=200"
              modbus_set_output_register("mensaje_mw10", 200)
              $ 1217 "Wait Continuar_M30=HI"
              while (modbus_get_signal_status("Continuar_M30") == False):
                sync()
              end
              $ 1218 "Wait: 1.0"
              sleep(1.0)
              $ 1219 "Set mensaje_mw10=150"
              modbus_set_output_register("mensaje_mw10", 150)
              $ 1220 "Wait: 1.0"
              sleep(1.0)
            end
            $ 1221 "MoveJ"
            $ 1222 "internos" "breakAfter"
            movej(internos, a=0.6981317007977318, v=0.5235987755982988)
            $ 1223 "Wait: 2.0"
            sleep(2.0)
            $ 1224 "If P1h[2]<P2h[2]"
            if (P1h[2]<P2h[2]):
              $ 1225 "acomodo≔(altura/(barrenosTotales-1))*(barrenoActual-1)"
              global acomodo=(altura/(barrenosTotales-1))*(barrenoActual-1)
              $ 1226 "tcp≔get_actual_tcp_pose()"
              global tcp= get_actual_tcp_pose ()
              $ 1227 "offset_altura≔p[tcp[0],tcp[1],((alta-0.0095)-(acomodo/1000)),tcp[3],tcp[4],tcp[5]]"
              global offset_altura=p[tcp[0],tcp[1],((alta-0.0095)-(acomodo/1000)),tcp[3],tcp[4],tcp[5]]
              $ 1228 "MoveL"
              $ 1229 "offset_altura" "breakAfter"
              movel(offset_altura, a=0.04, v=0.03)
            else:
              $ 1230 "Else" "noBreak"
              $ 1231 "acomodo≔(altura/(barrenosTotales-1))*(26-(barrenoActual-1))"
              global acomodo=(altura/(barrenosTotales-1))*(26-(barrenoActual-1))
              $ 1232 "tcp≔get_actual_tcp_pose()"
              global tcp= get_actual_tcp_pose ()
              $ 1233 "offset_altura≔p[tcp[0],tcp[1],((alta-0.0095)-(acomodo/1000)),tcp[3],tcp[4],tcp[5]]"
              global offset_altura=p[tcp[0],tcp[1],((alta-0.0095)-(acomodo/1000)),tcp[3],tcp[4],tcp[5]]
              $ 1234 "MoveL"
              $ 1235 "offset_altura" "breakAfter"
              movel(offset_altura, a=0.04, v=0.03)
            end
            $ 1236 "Freemove"
            $ 1237 "Wait: 2.0"
            sleep(2.0)
            $ 1238 "freedrive_mode()"
            freedrive_mode()
            $ 1239 "Wait: 2.5"
            sleep(2.5)
            $ 1240 "end_freedrive_mode()"
            end_freedrive_mode()
            $ 1241 "Wait: 0.3"
            sleep(0.3)
            $ 1242 "Set CO[1]=Encender"
            set_configurable_digital_out(1, True)
            $ 1243 "Wait: 1.0"
            sleep(1.0)
            $ 1244 "Wait: 0.3"
            sleep(0.3)
            $ 1245 "Wait: 0.3"
            sleep(0.3)
            $ 1246 "Wait: 0.3"
            sleep(0.3)
            $ 1247 "Loop 3 times"
            Loop_46 = 0
            while (Loop_46 < 3):
              $ 1248 "Poses_taladrado≔pose_sub(get_actual_tcp_pose(), bajada_broca)"
              global Poses_taladrado= pose_sub ( get_actual_tcp_pose (), bajada_broca)
              $ 1249 "Poses_taladrado" "breakAfter"
              movel(Poses_taladrado, a=0.005, v=0.001)
              $ 1250 "If bajada_broca≟p[0,0,0.018,0,0,0]"
              if (bajada_broca == p[0,0,0.018,0,0,0]):
                $ 1251 "num_barreno≔str_cat('Barreno: ',barrenoActual)"
                global num_barreno=str_cat("Barreno: ",barrenoActual)
                $ 1252 "tcp_actual≔get_actual_tcp_pose()"
                global tcp_actual= get_actual_tcp_pose ()
                $ 1253 "X_actual≔str_cat('     X: ',tcp_actual[0])"
                global X_actual=str_cat("     X: ",tcp_actual[0])
                $ 1254 "Y_actual≔str_cat('     Y: ',tcp_actual[1])"
                global Y_actual=str_cat("     Y: ",tcp_actual[1])
                $ 1255 "pos_barreno≔str_cat(X_actual,Y_actual)"
                global pos_barreno=str_cat(X_actual,Y_actual)
                $ 1256 "textmsg(num_barreno,pos_barreno)"
                textmsg(num_barreno,pos_barreno)
              end
              $ 1257 "Poses_taladrado≔pose_add(get_actual_tcp_pose(), bajada_broca)"
              global Poses_taladrado= pose_add ( get_actual_tcp_pose (), bajada_broca)
              $ 1258 "Poses_taladrado" "breakAfter"
              movel(Poses_taladrado, a=0.01, v=0.01)
              $ 1259 "bajada_broca≔pose_add(bajada_broca, p[0,0,0.006,0,0,0])"
              global bajada_broca= pose_add (bajada_broca, p[0,0,0.006,0,0,0])
              Loop_46 = Loop_46 + 1
            end
            $ 1260 "Direction: Base Z+"
            global move_thread_flag_1260=0
            thread move_thread_1260():
              enter_critical
              move_thread_flag_1260 = 1
              local towardsPos=calculate_point_to_move_towards(p[0.0,0.0,0.0,0.0,0.0,0.0], [0.0,0.0,1.0], 0.05)
              movel(towardsPos, a=0.04, v=0.03)
              move_thread_flag_1260 = 2
              exit_critical
            end
            move_thread_flag_1260 = 0
            move_thread_han_1260 = run move_thread_1260()
            while (True):
              sleep(1.0E-10)
              if (move_thread_flag_1260 > 1):
                join move_thread_han_1260
                $ 1261 "Until (distance)"
                break
              end
              sync()
            end
            $ 1262 "MoveJ"
            $ 1263 "internos" "breakAfter"
            movej(internos, a=0.6981317007977318, v=0.5235987755982988)
            $ 1264 "Wait: 0.3"
            sleep(0.3)
            $ 1265 "Set CO[1]=Apagar"
            set_configurable_digital_out(1, False)
            $ 1266 "Wait: 0.3"
            sleep(0.3)
            $ 1267 "If barrenoActual≟13"
            if (barrenoActual == 13):
              $ 1268 "Direction: Base Z+"
              global move_thread_flag_1268=0
              thread move_thread_1268():
                enter_critical
                move_thread_flag_1268 = 1
                local towardsPos=calculate_point_to_move_towards(p[0.0,0.0,0.0,0.0,0.0,0.0], [0.0,0.0,1.0], 0.03)
                movel(towardsPos, a=1.2, v=0.25)
                move_thread_flag_1268 = 2
                exit_critical
              end
              move_thread_flag_1268 = 0
              move_thread_han_1268 = run move_thread_1268()
              while (True):
                sleep(1.0E-10)
                if (move_thread_flag_1268 > 1):
                  join move_thread_han_1268
                  $ 1269 "Until (distance)"
                  break
                end
                sync()
              end
              $ 1270 "MoveJ"
              $ 1271 "Zona_der1" "breakAfter"
              movej(get_inverse_kin(Zona_der1_p, qnear=Zona_der1_q), a=1.3962634015954636, v=1.0471975511965976)
              $ 1272 "Posicion_Cero" "breakAfter"
              movej(get_inverse_kin(Posicion_Cero_p, qnear=Posicion_Cero_q), a=1.3962634015954636, v=1.0471975511965976)
              $ 1273 "Call Quitar_Broca_Chida"
              Quitar_Broca_Chida()
              $ 1274 "Call Poner_Broca"
              Poner_Broca()
              $ 1275 "MoveJ"
              $ 1276 "Posicion_Cero" "breakAfter"
              movej(get_inverse_kin(Posicion_Cero_p, qnear=Posicion_Cero_q), a=1.3962634015954636, v=1.0471975511965976)
              $ 1277 "Zona_der1" "breakAfter"
              movej(get_inverse_kin(Zona_der1_p, qnear=Zona_der1_q), a=1.3962634015954636, v=1.0471975511965976)
            else:
              $ 1278 "ElseIf barrenoActual≟27"
              if (barrenoActual == 27):
                $ 1279 "Direction: Base Z+"
                global move_thread_flag_1279=0
                thread move_thread_1279():
                  enter_critical
                  move_thread_flag_1279 = 1
                  local towardsPos=calculate_point_to_move_towards(p[0.0,0.0,0.0,0.0,0.0,0.0], [0.0,0.0,1.0], 0.03)
                  movel(towardsPos, a=1.2, v=0.25)
                  move_thread_flag_1279 = 2
                  exit_critical
                end
                move_thread_flag_1279 = 0
                move_thread_han_1279 = run move_thread_1279()
                while (True):
                  sleep(1.0E-10)
                  if (move_thread_flag_1279 > 1):
                    join move_thread_han_1279
                    $ 1280 "Until (distance)"
                    break
                  end
                  sync()
                end
                $ 1281 "MoveJ"
                $ 1282 "Zona_der1" "breakAfter"
                movej(get_inverse_kin(Zona_der1_p, qnear=Zona_der1_q), a=1.3962634015954636, v=1.0471975511965976)
                $ 1283 "Posicion_Cero" "breakAfter"
                movej(get_inverse_kin(Posicion_Cero_p, qnear=Posicion_Cero_q), a=1.3962634015954636, v=1.0471975511965976)
                $ 1284 "Call Quitar_Broca_Chida"
                Quitar_Broca_Chida()
                $ 1285 "Set carrusel_home=Encender"
                modbus_set_output_signal("carrusel_home", True)
                $ 1286 "Wait: 1.0"
                sleep(1.0)
                $ 1287 "Set carrusel_home=Apagar"
                modbus_set_output_signal("carrusel_home", False)
                $ 1288 "Set mensaje_mw10=70"
                modbus_set_output_register("mensaje_mw10", 70)
                $ 1289 "Wait Continuar_M30=HI"
                while (modbus_get_signal_status("Continuar_M30") == False):
                  sync()
                end
                $ 1290 "Wait: 1.0"
                sleep(1.0)
                $ 1291 "Set mensaje_mw10=120"
                modbus_set_output_register("mensaje_mw10", 120)
                $ 1292 "Wait Continuar_M30=HI"
                while (modbus_get_signal_status("Continuar_M30") == False):
                  sync()
                end
                $ 1293 "Wait: 1.0"
                sleep(1.0)
                $ 1294 "Set carrusel_home=Encender"
                modbus_set_output_signal("carrusel_home", True)
                $ 1295 "Wait: 1.0"
                sleep(1.0)
                $ 1296 "Set carrusel_home=Apagar"
                modbus_set_output_signal("carrusel_home", False)
                $ 1297 "Set mensaje_mw10=75"
                modbus_set_output_register("mensaje_mw10", 75)
                $ 1298 "Wait Continuar_M30=HI"
                while (modbus_get_signal_status("Continuar_M30") == False):
                  sync()
                end
                $ 1299 "Wait: 1.0"
                sleep(1.0)
                $ 1300 "Call Poner_Broca"
                Poner_Broca()
                $ 1301 "broca≔1935"
                global broca=1935
                $ 1302 "MoveJ"
                $ 1303 "Posicion_Cero" "breakAfter"
                movej(get_inverse_kin(Posicion_Cero_p, qnear=Posicion_Cero_q), a=1.3962634015954636, v=1.0471975511965976)
                $ 1304 "Zona_der1" "breakAfter"
                movej(get_inverse_kin(Zona_der1_p, qnear=Zona_der1_q), a=1.3962634015954636, v=1.0471975511965976)
                $ 1305 "Set mensaje_mw10=80"
                modbus_set_output_register("mensaje_mw10", 80)
                $ 1306 "Wait Continuar_M30=HI"
                while (modbus_get_signal_status("Continuar_M30") == False):
                  sync()
                end
                $ 1307 "Wait: 1.0"
                sleep(1.0)
                $ 1308 "Set mensaje_mw10=150"
                modbus_set_output_register("mensaje_mw10", 150)
                $ 1309 "Wait Continuar_M30=HI"
                while (modbus_get_signal_status("Continuar_M30") == False):
                  sync()
                end
                $ 1310 "Wait: 1.0"
                sleep(1.0)
              end
            end
            $ 1311 "barrenoActual≔barrenoActual+1"
            global barrenoActual=barrenoActual+1
          end
          $ 1312 "Linea 1 a 1935"
          $ 1313 "broca≔1935"
          global broca=1935
          $ 1314 "Buje_inicial"
          $ 1315 "Buje_Inicial≔L1B2"
          global Buje_Inicial=L1B2
          $ 1316 "Buje_final"
          $ 1317 "Buje_Final≔L1B1"
          global Buje_Final=L1B1
          $ 1318 "barrenosTotales≔27"
          global barrenosTotales=27
          $ 1319 "barrenoActual≔1"
          global barrenoActual=1
          $ 1320 "Loop barrenoActual≤barrenosTotales"
          while (barrenoActual <= barrenosTotales):
            $ 1321 "MoveL"
            $ 1322 "bajada_broca≔p[0,0,0.009,0,0,0]"
            global bajada_broca=p[0,0,0.009,0,0,0]
            $ 1323 "internos≔interpolate_pose(Buje_Inicial, Buje_Final, ((barrenoActual)-1)/((barrenosTotales)-1))"
            global internos= interpolate_pose (Buje_Inicial, Buje_Final, ((barrenoActual)-1)/((barrenosTotales)-1))
            $ 1324 "Alturas"
            $ 1325 "If barrenoActual≟1 or barrenoActual≟3 or barrenoActual≟5 or barrenoActual≟7 or barrenoActual≟9 or barrenoActual≟11 or barrenoActual≟13 or barrenoActual≟15 or barrenoActual≟17 or barrenoActual≟19 or barrenoActual≟21 or barrenoActual≟23 or barrenoActual≟25 or barrenoActual≟27"
            if (barrenoActual == 1  or  barrenoActual == 3  or  barrenoActual == 5  or  barrenoActual == 7  or  barrenoActual == 9  or  barrenoActual == 11  or  barrenoActual == 13  or  barrenoActual == 15  or  barrenoActual == 17  or  barrenoActual == 19  or  barrenoActual == 21  or  barrenoActual == 23  or  barrenoActual == 25  or  barrenoActual == 27):
              $ 1326 "Set mensaje_mw10=200"
              modbus_set_output_register("mensaje_mw10", 200)
              $ 1327 "Wait Continuar_M30=HI"
              while (modbus_get_signal_status("Continuar_M30") == False):
                sync()
              end
              $ 1328 "Wait: 1.0"
              sleep(1.0)
              $ 1329 "Set mensaje_mw10=150"
              modbus_set_output_register("mensaje_mw10", 150)
              $ 1330 "Wait: 1.0"
              sleep(1.0)
            end
            $ 1331 "MoveJ"
            $ 1332 "internos" "breakAfter"
            movej(internos, a=0.6981317007977318, v=0.5235987755982988)
            $ 1333 "Wait: 2.0"
            sleep(2.0)
            $ 1334 "If P1h[2]<P2h[2]"
            if (P1h[2]<P2h[2]):
              $ 1335 "acomodo≔(altura/(barrenosTotales-1))*(barrenoActual-1)"
              global acomodo=(altura/(barrenosTotales-1))*(barrenoActual-1)
              $ 1336 "tcp≔get_actual_tcp_pose()"
              global tcp= get_actual_tcp_pose ()
              $ 1337 "offset_altura≔p[tcp[0],tcp[1],((alta-0.0095)-(acomodo/1000)),tcp[3],tcp[4],tcp[5]]"
              global offset_altura=p[tcp[0],tcp[1],((alta-0.0095)-(acomodo/1000)),tcp[3],tcp[4],tcp[5]]
              $ 1338 "MoveL"
              $ 1339 "offset_altura" "breakAfter"
              movel(offset_altura, a=0.04, v=0.03)
            else:
              $ 1340 "Else" "noBreak"
              $ 1341 "acomodo≔(altura/(barrenosTotales-1))*(26-(barrenoActual-1))"
              global acomodo=(altura/(barrenosTotales-1))*(26-(barrenoActual-1))
              $ 1342 "tcp≔get_actual_tcp_pose()"
